LIN {X 69.907,Y 96.272,Z 65.686,A 180.000,B 0.000,C 180.000} C_DIS
LIN {X 69.876,Y 96.200,Z 65.684,A 180.000,B 0.000,C 180.000} C_DIS
LIN {X 69.842,Y 96.129,Z 65.681,A 180.000,B 0.000,C 180.000} C_DIS
LIN {X 69.807,Y 96.058,Z 65.678,A 180.000,B 0.000,C 180.000} C_DIS
LIN {X 69.735,Y 95.918,Z 65.673,A 180.000,B 0.000,C 180.000} C_DIS
LIN {X 69.664,Y 95.778,Z 65.668,A 180.000,B 0.000,C 180.000} C_DIS
LIN {X 69.628,Y 95.707,Z 65.665,A 180.000,B 0.000,C 180.000} C_DIS
LIN {X 69.592,Y 95.637,Z 65.662,A 180.000,B 0.000,C 180.000} C_DIS
LIN {X 69.557,Y 95.567,Z 65.660,A 180.000,B 0.000,C 180.000} C_DIS
LIN {X 69.521,Y 95.497,Z 65.657,A 180.000,B 0.000,C 180.000} C_DIS
LIN {X 69.483,Y 95.428,Z 65.655,A 180.000,B 0.000,C 180.000} C_DIS
LIN {X 69.443,Y 95.360,Z 65.652,A 180.000,B 0.000,C 180.000} C_DIS
LIN {X 69.403,Y 95.292,Z 65.650,A 180.000,B 0.000,C 180.000} C_DIS
LIN {X 69.323,Y 95.156,Z 65.645,A 180.000,B 0.000,C 180.000} C_DIS
LIN {X 69.243,Y 95.021,Z 65.640,A 180.000,B 0.000,C 180.000} C_DIS
LIN {X 69.163,Y 94.885,Z 65.635,A 180.000,B 0.000,C 180.000} C_DIS
LIN {X 69.081,Y 94.751,Z 65.630,A 180.000,B 0.000,C 180.000} C_DIS
LIN {X 68.992,Y 94.620,Z 65.625,A 180.000,B 0.000,C 180.000} C_DIS
LIN {X 68.904,Y 94.490,Z 65.621,A 180.000,B 0.000,C 180.000} C_DIS
LIN {X 68.815,Y 94.360,Z 65.616,A 180.000,B 0.000,C 180.000} C_DIS
LIN {X 68.727,Y 94.230,Z 65.612,A 180.000,B 0.000,C 180.000} C_DIS
LIN {X 68.636,Y 94.101,Z 65.607,A 180.000,B 0.000,C 180.000} C_DIS
LIN {X 68.540,Y 93.976,Z 65.603,A 180.000,B 0.000,C 180.000} C_DIS
LIN {X 68.444,Y 93.851,Z 65.598,A 180.000,B 0.000,C 180.000} C_DIS
LIN {X 68.347,Y 93.727,Z 65.594,A 180.000,B 0.000,C 180.000} C_DIS
LIN {X 68.251,Y 93.603,Z 65.590,A 180.000,B 0.000,C 180.000} C_DIS
LIN {X 68.152,Y 93.479,Z 65.586,A 180.000,B 0.000,C 180.000} C_DIS
LIN {X 68.049,Y 93.361,Z 65.582,A 180.000,B 0.000,C 180.000} C_DIS
LIN {X 67.945,Y 93.243,Z 65.578,A 180.000,B 0.000,C 180.000} C_DIS
LIN {X 67.840,Y 93.125,Z 65.574,A 180.000,B 0.000,C 180.000} C_DIS
LIN {X 67.736,Y 93.007,Z 65.571,A 180.000,B 0.000,C 180.000} C_DIS
LIN {X 67.630,Y 92.890,Z 65.567,A 180.000,B 0.000,C 180.000} C_DIS
LIN {X 67.519,Y 92.778,Z 65.563,A 180.000,B 0.000,C 180.000} C_DIS
LIN {X 67.408,Y 92.667,Z 65.560,A 180.000,B 0.000,C 180.000} C_DIS
LIN {X 67.297,Y 92.555,Z 65.556,A 180.000,B 0.000,C 180.000} C_DIS
LIN {X 67.185,Y 92.444,Z 65.553,A 180.000,B 0.000,C 180.000} C_DIS
LIN {X 67.072,Y 92.334,Z 65.550,A 180.000,B 0.000,C 180.000} C_DIS
LIN {X 66.955,Y 92.230,Z 65.547,A 180.000,B 0.000,C 180.000} C_DIS
LIN {X 66.837,Y 92.125,Z 65.544,A 180.000,B 0.000,C 180.000} C_DIS
LIN {X 66.718,Y 92.021,Z 65.541,A 180.000,B 0.000,C 180.000} C_DIS
LIN {X 66.600,Y 91.917,Z 65.538,A 180.000,B 0.000,C 180.000} C_DIS
LIN {X 66.481,Y 91.815,Z 65.535,A 180.000,B 0.000,C 180.000} C_DIS
LIN {X 66.357,Y 91.718,Z 65.532,A 180.000,B 0.000,C 180.000} C_DIS
LIN {X 66.232,Y 91.621,Z 65.530,A 180.000,B 0.000,C 180.000} C_DIS
LIN {X 66.108,Y 91.524,Z 65.527,A 180.000,B 0.000,C 180.000} C_DIS
LIN {X 65.858,Y 91.333,Z 65.523,A 180.000,B 0.000,C 180.000} C_DIS
LIN {X 65.597,Y 91.156,Z 65.518,A 180.000,B 0.000,C 180.000} C_DIS
LIN {X 65.337,Y 90.978,Z 65.515,A 180.000,B 0.000,C 180.000} C_DIS
LIN {X 65.070,Y 90.811,Z 65.511,A 180.000,B 0.000,C 180.000} C_DIS
LIN {X 64.799,Y 90.651,Z 65.508,A 180.000,B 0.000,C 180.000} C_DIS
LIN {X 64.527,Y 90.492,Z 65.506,A 180.000,B 0.000,C 180.000} C_DIS
LIN {X 64.247,Y 90.348,Z 65.504,A 180.000,B 0.000,C 180.000} C_DIS
LIN {X 63.966,Y 90.205,Z 65.502,A 180.000,B 0.000,C 180.000} C_DIS
LIN {X 63.680,Y 90.072,Z 65.501,A 180.000,B 0.000,C 180.000} C_DIS
LIN {X 63.391,Y 89.947,Z 65.500,A 180.000,B 0.000,C 180.000} C_DIS
LIN {X 63.141,Y 89.840,Z 65.500,A 180.000,B 0.000,C 180.000} C_DIS
; Cutting Move Starts
LIN {X 63.109,Y 89.827,Z 65.500,A 180.000,B 0.000,C 180.000} C_DIS
LIN {X 62.930,Y 89.762,Z 65.500,A 180.000,B 0.000,C 180.000} C_DIS
LIN {X 62.573,Y 89.633,Z 65.500,A 180.000,B 0.000,C 180.000} C_DIS
LIN {X 62.394,Y 89.569,Z 65.500,A 180.000,B 0.000,C 180.000} C_DIS
LIN {X 62.387,Y 89.567,Z 65.500,A 180.000,B 0.000,C 180.000} C_DIS
LIN {X 62.215,Y 89.516,Z 65.500,A 180.000,B 0.000,C 180.000} C_DIS
LIN {X 61.777,Y 89.388,Z 65.500,A 180.000,B 0.000,C 180.000} C_DIS
LIN {X 61.679,Y 89.360,Z 65.500,A 180.000,B 0.000,C 180.000} C_DIS
LIN {X 61.500,Y 89.316,Z 65.500,A 180.000,B 0.000,C 180.000} C_DIS
LIN {X 60.964,Y 89.196,Z 65.500,A 180.000,B 0.000,C 180.000} C_DIS
LIN {X 60.785,Y 89.161,Z 65.500,A 180.000,B 0.000,C 180.000} C_DIS
LIN {X 60.606,Y 89.132,Z 65.500,A 180.000,B 0.000,C 180.000} C_DIS
LIN {X 60.249,Y 89.076,Z 65.500,A 180.000,B 0.000,C 180.000} C_DIS
LIN {X 60.070,Y 89.049,Z 65.500,A 180.000,B 0.000,C 180.000} C_DIS
LIN {X 59.892,Y 89.031,Z 65.500,A 180.000,B 0.000,C 180.000} C_DIS
LIN {X 59.534,Y 88.997,Z 65.500,A 180.000,B 0.000,C 180.000} C_DIS
LIN {X 59.355,Y 88.980,Z 65.500,A 180.000,B 0.000,C 180.000} C_DIS
LIN {X 59.176,Y 88.970,Z 65.500,A 180.000,B 0.000,C 180.000} C_DIS
LIN {X 58.640,Y 88.953,Z 65.500,A 180.000,B 0.000,C 180.000} C_DIS
LIN {X 58.461,Y 88.950,Z 65.500,A 180.000,B 0.000,C 180.000} C_DIS
LIN {X 58.282,Y 88.956,Z 65.500,A 180.000,B 0.000,C 180.000} C_DIS
LIN {X 57.925,Y 88.967,Z 65.500,A 180.000,B 0.000,C 180.000} C_DIS
LIN {X 57.746,Y 88.973,Z 65.500,A 180.000,B 0.000,C 180.000} C_DIS
LIN {X 57.567,Y 88.987,Z 65.500,A 180.000,B 0.000,C 180.000} C_DIS
LIN {X 57.031,Y 89.038,Z 65.500,A 180.000,B 0.000,C 180.000} C_DIS
LIN {X 56.852,Y 89.060,Z 65.500,A 180.000,B 0.000,C 180.000} C_DIS
LIN {X 56.316,Y 89.145,Z 65.500,A 180.000,B 0.000,C 180.000} C_DIS
LIN {X 56.137,Y 89.174,Z 65.500,A 180.000,B 0.000,C 180.000} C_DIS
LIN {X 55.977,Y 89.209,Z 65.500,A 180.000,B 0.000,C 180.000} C_DIS
LIN {X 55.601,Y 89.293,Z 65.500,A 180.000,B 0.000,C 180.000} C_DIS
LIN {X 55.422,Y 89.334,Z 65.500,A 180.000,B 0.000,C 180.000} C_DIS
LIN {X 55.243,Y 89.382,Z 65.500,A 180.000,B 0.000,C 180.000} C_DIS
LIN {X 54.707,Y 89.538,Z 65.500,A 180.000,B 0.000,C 180.000} C_DIS
LIN {X 54.613,Y 89.567,Z 65.500,A 180.000,B 0.000,C 180.000} C_DIS
LIN {X 54.528,Y 89.597,Z 65.500,A 180.000,B 0.000,C 180.000} C_DIS
LIN {X 53.992,Y 89.790,Z 65.500,A 180.000,B 0.000,C 180.000} C_DIS
LIN {X 53.813,Y 89.859,Z 65.500,A 180.000,B 0.000,C 180.000} C_DIS
LIN {X 53.455,Y 90.014,Z 65.500,A 180.000,B 0.000,C 180.000} C_DIS
LIN {X 53.248,Y 90.103,Z 65.500,A 180.000,B 0.000,C 180.000} C_DIS
LIN {X 53.098,Y 90.173,Z 65.500,A 180.000,B 0.000,C 180.000} C_DIS
LIN {X 52.919,Y 90.264,Z 65.500,A 180.000,B 0.000,C 180.000} C_DIS
LIN {X 52.533,Y 90.461,Z 65.500,A 180.000,B 0.000,C 180.000} C_DIS
LIN {X 52.383,Y 90.543,Z 65.500,A 180.000,B 0.000,C 180.000} C_DIS
LIN {X 51.847,Y 90.860,Z 65.500,A 180.000,B 0.000,C 180.000} C_DIS
LIN {X 51.668,Y 90.975,Z 65.500,A 180.000,B 0.000,C 180.000} C_DIS
LIN {X 51.310,Y 91.218,Z 65.500,A 180.000,B 0.000,C 180.000} C_DIS
LIN {X 51.131,Y 91.341,Z 65.500,A 180.000,B 0.000,C 180.000} C_DIS
LIN {X 51.113,Y 91.355,Z 65.500,A 180.000,B 0.000,C 180.000} C_DIS
LIN {X 50.953,Y 91.478,Z 65.500,A 180.000,B 0.000,C 180.000} C_DIS
LIN {X 50.595,Y 91.755,Z 65.500,A 180.000,B 0.000,C 180.000} C_DIS
LIN {X 50.429,Y 91.891,Z 65.500,A 180.000,B 0.000,C 180.000} C_DIS
LIN {X 50.024,Y 92.249,Z 65.500,A 180.000,B 0.000,C 180.000} C_DIS
LIN {X 49.880,Y 92.379,Z 65.500,A 180.000,B 0.000,C 180.000} C_DIS
LIN {X 49.831,Y 92.427,Z 65.500,A 180.000,B 0.000,C 180.000} C_DIS
LIN {X 49.474,Y 92.785,Z 65.500,A 180.000,B 0.000,C 180.000} C_DIS
LIN {X 49.344,Y 92.917,Z 65.500,A 180.000,B 0.000,C 180.000} C_DIS
LIN {X 49.302,Y 92.964,Z 65.500,A 180.000,B 0.000,C 180.000} C_DIS
LIN {X 48.986,Y 93.321,Z 65.500,A 180.000,B 0.000,C 180.000} C_DIS
LIN {X 48.830,Y 93.500,Z 65.500,A 180.000,B 0.000,C 180.000} C_DIS
LIN {X 48.807,Y 93.528,Z 65.500,A 180.000,B 0.000,C 180.000} C_DIS
LIN {X 48.690,Y 93.679,Z 65.500,A 180.000,B 0.000,C 180.000} C_DIS
LIN {X 48.413,Y 94.036,Z 65.500,A 180.000,B 0.000,C 180.000} C_DIS
LIN {X 48.283,Y 94.215,Z 65.500,A 180.000,B 0.000,C 180.000} C_DIS
LIN {X 48.040,Y 94.573,Z 65.500,A 180.000,B 0.000,C 180.000} C_DIS
LIN {X 47.919,Y 94.751,Z 65.500,A 180.000,B 0.000,C 180.000} C_DIS
LIN {X 47.914,Y 94.760,Z 65.500,A 180.000,B 0.000,C 180.000} C_DIS
LIN {X 47.811,Y 94.930,Z 65.500,A 180.000,B 0.000,C 180.000} C_DIS
LIN {X 47.556,Y 95.361,Z 65.500,A 180.000,B 0.000,C 180.000} C_DIS
LIN {X 47.496,Y 95.466,Z 65.500,A 180.000,B 0.000,C 180.000} C_DIS
LIN {X 47.404,Y 95.645,Z 65.500,A 180.000,B 0.000,C 180.000} C_DIS
LIN {X 47.198,Y 96.048,Z 65.500,A 180.000,B 0.000,C 180.000} C_DIS
LIN {X 47.133,Y 96.181,Z 65.500,A 180.000,B 0.000,C 180.000} C_DIS
LIN {X 47.055,Y 96.360,Z 65.500,A 180.000,B 0.000,C 180.000} C_DIS
LIN {X 46.900,Y 96.718,Z 65.500,A 180.000,B 0.000,C 180.000} C_DIS
LIN {X 46.841,Y 96.856,Z 65.500,A 180.000,B 0.000,C 180.000} C_DIS
LIN {X 46.825,Y 96.897,Z 65.500,A 180.000,B 0.000,C 180.000} C_DIS
LIN {X 46.760,Y 97.075,Z 65.500,A 180.000,B 0.000,C 180.000} C_DIS
LIN {X 46.631,Y 97.433,Z 65.500,A 180.000,B 0.000,C 180.000} C_DIS
LIN {X 46.568,Y 97.612,Z 65.500,A 180.000,B 0.000,C 180.000} C_DIS
LIN {X 46.514,Y 97.790,Z 65.500,A 180.000,B 0.000,C 180.000} C_DIS
LIN {X 46.410,Y 98.148,Z 65.500,A 180.000,B 0.000,C 180.000} C_DIS
LIN {X 46.358,Y 98.327,Z 65.500,A 180.000,B 0.000,C 180.000} C_DIS
LIN {X 46.315,Y 98.505,Z 65.500,A 180.000,B 0.000,C 180.000} C_DIS
LIN {X 46.195,Y 99.042,Z 65.500,A 180.000,B 0.000,C 180.000} C_DIS
LIN {X 46.160,Y 99.221,Z 65.500,A 180.000,B 0.000,C 180.000} C_DIS
LIN {X 46.126,Y 99.434,Z 65.500,A 180.000,B 0.000,C 180.000} C_DIS
LIN {X 46.075,Y 99.757,Z 65.500,A 180.000,B 0.000,C 180.000} C_DIS
LIN {X 46.048,Y 99.936,Z 65.500,A 180.000,B 0.000,C 180.000} C_DIS
LIN {X 46.030,Y 100.114,Z 65.500,A 180.000,B 0.000,C 180.000} C_DIS
LIN {X 45.996,Y 100.472,Z 65.500,A 180.000,B 0.000,C 180.000} C_DIS
LIN {X 45.979,Y 100.651,Z 65.500,A 180.000,B 0.000,C 180.000} C_DIS
LIN {X 45.970,Y 100.829,Z 65.500,A 180.000,B 0.000,C 180.000} C_DIS
LIN {X 45.953,Y 101.366,Z 65.500,A 180.000,B 0.000,C 180.000} C_DIS
LIN {X 45.950,Y 101.545,Z 65.500,A 180.000,B 0.000,C 180.000} C_DIS
LIN {X 45.956,Y 101.723,Z 65.500,A 180.000,B 0.000,C 180.000} C_DIS
LIN {X 45.967,Y 102.081,Z 65.500,A 180.000,B 0.000,C 180.000} C_DIS
LIN {X 45.973,Y 102.260,Z 65.500,A 180.000,B 0.000,C 180.000} C_DIS
LIN {X 45.988,Y 102.438,Z 65.500,A 180.000,B 0.000,C 180.000} C_DIS
LIN {X 46.038,Y 102.975,Z 65.500,A 180.000,B 0.000,C 180.000} C_DIS
LIN {X 46.060,Y 103.153,Z 65.500,A 180.000,B 0.000,C 180.000} C_DIS
LIN {X 46.145,Y 103.690,Z 65.500,A 180.000,B 0.000,C 180.000} C_DIS
LIN {X 46.176,Y 103.869,Z 65.500,A 180.000,B 0.000,C 180.000} C_DIS
LIN {X 46.215,Y 104.047,Z 65.500,A 180.000,B 0.000,C 180.000} C_DIS
LIN {X 46.305,Y 104.449,Z 65.500,A 180.000,B 0.000,C 180.000} C_DIS
LIN {X 46.335,Y 104.584,Z 65.500,A 180.000,B 0.000,C 180.000} C_DIS
LIN {X 46.384,Y 104.762,Z 65.500,A 180.000,B 0.000,C 180.000} C_DIS
LIN {X 46.540,Y 105.299,Z 65.500,A 180.000,B 0.000,C 180.000} C_DIS
LIN {X 46.599,Y 105.477,Z 65.500,A 180.000,B 0.000,C 180.000} C_DIS
LIN {X 46.792,Y 106.014,Z 65.500,A 180.000,B 0.000,C 180.000} C_DIS
LIN {X 46.841,Y 106.144,Z 65.500,A 180.000,B 0.000,C 180.000} C_DIS
LIN {X 46.861,Y 106.193,Z 65.500,A 180.000,B 0.000,C 180.000} C_DIS
LIN {X 47.093,Y 106.729,Z 65.500,A 180.000,B 0.000,C 180.000} C_DIS
LIN {X 47.176,Y 106.908,Z 65.500,A 180.000,B 0.000,C 180.000} C_DIS
LIN {X 47.198,Y 106.952,Z 65.500,A 180.000,B 0.000,C 180.000} C_DIS
LIN {X 47.449,Y 107.444,Z 65.500,A 180.000,B 0.000,C 180.000} C_DIS
LIN {X 47.546,Y 107.623,Z 65.500,A 180.000,B 0.000,C 180.000} C_DIS
LIN {X 47.863,Y 108.159,Z 65.500,A 180.000,B 0.000,C 180.000} C_DIS
LIN {X 47.914,Y 108.240,Z 65.500,A 180.000,B 0.000,C 180.000} C_DIS
LIN {X 47.979,Y 108.338,Z 65.500,A 180.000,B 0.000,C 180.000} C_DIS
LIN {X 48.271,Y 108.767,Z 65.500,A 180.000,B 0.000,C 180.000} C_DIS
LIN {X 48.345,Y 108.874,Z 65.500,A 180.000,B 0.000,C 180.000} C_DIS
LIN {X 48.450,Y 109.012,Z 65.500,A 180.000,B 0.000,C 180.000} C_DIS
LIN {X 48.759,Y 109.410,Z 65.500,A 180.000,B 0.000,C 180.000} C_DIS
LIN {X 48.807,Y 109.472,Z 65.500,A 180.000,B 0.000,C 180.000} C_DIS
LIN {X 48.907,Y 109.589,Z 65.500,A 180.000,B 0.000,C 180.000} C_DIS
LIN {X 49.223,Y 109.947,Z 65.500,A 180.000,B 0.000,C 180.000} C_DIS
LIN {X 49.344,Y 110.083,Z 65.500,A 180.000,B 0.000,C 180.000} C_DIS
LIN {X 49.384,Y 110.126,Z 65.500,A 180.000,B 0.000,C 180.000} C_DIS
LIN {X 49.523,Y 110.264,Z 65.500,A 180.000,B 0.000,C 180.000} C_DIS
LIN {X 49.742,Y 110.483,Z 65.500,A 180.000,B 0.000,C 180.000} C_DIS
LIN {X 49.880,Y 110.621,Z 65.500,A 180.000,B 0.000,C 180.000} C_DIS
LIN {X 49.923,Y 110.662,Z 65.500,A 180.000,B 0.000,C 180.000} C_DIS
LIN {X 50.059,Y 110.782,Z 65.500,A 180.000,B 0.000,C 180.000} C_DIS
LIN {X 50.416,Y 111.098,Z 65.500,A 180.000,B 0.000,C 180.000} C_DIS
LIN {X 50.535,Y 111.198,Z 65.500,A 180.000,B 0.000,C 180.000} C_DIS
LIN {X 50.595,Y 111.245,Z 65.500,A 180.000,B 0.000,C 180.000} C_DIS
LIN {X 50.996,Y 111.556,Z 65.500,A 180.000,B 0.000,C 180.000} C_DIS
LIN {X 51.131,Y 111.659,Z 65.500,A 180.000,B 0.000,C 180.000} C_DIS
LIN {X 51.241,Y 111.734,Z 65.500,A 180.000,B 0.000,C 180.000} C_DIS
LIN {X 51.668,Y 112.025,Z 65.500,A 180.000,B 0.000,C 180.000} C_DIS
LIN {X 51.769,Y 112.092,Z 65.500,A 180.000,B 0.000,C 180.000} C_DIS
LIN {X 51.847,Y 112.140,Z 65.500,A 180.000,B 0.000,C 180.000} C_DIS
LIN {X 52.383,Y 112.457,Z 65.500,A 180.000,B 0.000,C 180.000} C_DIS
LIN {X 52.562,Y 112.554,Z 65.500,A 180.000,B 0.000,C 180.000} C_DIS
LIN {X 53.059,Y 112.807,Z 65.500,A 180.000,B 0.000,C 180.000} C_DIS
LIN {X 53.098,Y 112.827,Z 65.500,A 180.000,B 0.000,C 180.000} C_DIS
LIN {X 53.277,Y 112.909,Z 65.500,A 180.000,B 0.000,C 180.000} C_DIS
LIN {X 53.813,Y 113.141,Z 65.500,A 180.000,B 0.000,C 180.000} C_DIS
LIN {X 53.870,Y 113.165,Z 65.500,A 180.000,B 0.000,C 180.000} C_DIS
LIN {X 53.992,Y 113.210,Z 65.500,A 180.000,B 0.000,C 180.000} C_DIS
LIN {X 54.528,Y 113.403,Z 65.500,A 180.000,B 0.000,C 180.000} C_DIS
LIN {X 54.707,Y 113.462,Z 65.500,A 180.000,B 0.000,C 180.000} C_DIS
LIN {X 55.243,Y 113.618,Z 65.500,A 180.000,B 0.000,C 180.000} C_DIS
LIN {X 55.422,Y 113.666,Z 65.500,A 180.000,B 0.000,C 180.000} C_DIS
LIN {X 55.575,Y 113.701,Z 65.500,A 180.000,B 0.000,C 180.000} C_DIS
LIN {X 55.958,Y 113.786,Z 65.500,A 180.000,B 0.000,C 180.000} C_DIS
LIN {X 56.056,Y 113.808,Z 65.500,A 180.000,B 0.000,C 180.000} C_DIS
LIN {X 56.137,Y 113.826,Z 65.500,A 180.000,B 0.000,C 180.000} C_DIS
LIN {X 56.316,Y 113.855,Z 65.500,A 180.000,B 0.000,C 180.000} C_DIS
LIN {X 56.852,Y 113.940,Z 65.500,A 180.000,B 0.000,C 180.000} C_DIS
LIN {X 57.031,Y 113.962,Z 65.500,A 180.000,B 0.000,C 180.000} C_DIS
LIN {X 57.567,Y 114.013,Z 65.500,A 180.000,B 0.000,C 180.000} C_DIS
LIN {X 57.746,Y 114.027,Z 65.500,A 180.000,B 0.000,C 180.000} C_DIS
LIN {X 57.925,Y 114.033,Z 65.500,A 180.000,B 0.000,C 180.000} C_DIS
LIN {X 58.282,Y 114.044,Z 65.500,A 180.000,B 0.000,C 180.000} C_DIS
LIN {X 58.461,Y 114.050,Z 65.500,A 180.000,B 0.000,C 180.000} C_DIS
LIN {X 58.640,Y 114.047,Z 65.500,A 180.000,B 0.000,C 180.000} C_DIS
LIN {X 59.176,Y 114.030,Z 65.500,A 180.000,B 0.000,C 180.000} C_DIS
LIN {X 59.355,Y 114.020,Z 65.500,A 180.000,B 0.000,C 180.000} C_DIS
LIN {X 59.534,Y 114.003,Z 65.500,A 180.000,B 0.000,C 180.000} C_DIS
LIN {X 59.891,Y 113.969,Z 65.500,A 180.000,B 0.000,C 180.000} C_DIS
LIN {X 60.070,Y 113.951,Z 65.500,A 180.000,B 0.000,C 180.000} C_DIS
LIN {X 60.249,Y 113.924,Z 65.500,A 180.000,B 0.000,C 180.000} C_DIS
LIN {X 60.606,Y 113.868,Z 65.500,A 180.000,B 0.000,C 180.000} C_DIS
LIN {X 60.785,Y 113.839,Z 65.500,A 180.000,B 0.000,C 180.000} C_DIS
LIN {X 60.964,Y 113.804,Z 65.500,A 180.000,B 0.000,C 180.000} C_DIS
LIN {X 61.500,Y 113.684,Z 65.500,A 180.000,B 0.000,C 180.000} C_DIS
LIN {X 61.679,Y 113.640,Z 65.500,A 180.000,B 0.000,C 180.000} C_DIS
LIN {X 61.858,Y 113.588,Z 65.500,A 180.000,B 0.000,C 180.000} C_DIS
LIN {X 62.215,Y 113.484,Z 65.500,A 180.000,B 0.000,C 180.000} C_DIS
LIN {X 62.394,Y 113.431,Z 65.500,A 180.000,B 0.000,C 180.000} C_DIS
LIN {X 62.573,Y 113.367,Z 65.500,A 180.000,B 0.000,C 180.000} C_DIS
LIN {X 62.930,Y 113.238,Z 65.500,A 180.000,B 0.000,C 180.000} C_DIS
LIN {X 63.109,Y 113.173,Z 65.500,A 180.000,B 0.000,C 180.000} C_DIS
LIN {X 63.130,Y 113.165,Z 65.500,A 180.000,B 0.000,C 180.000} C_DIS
LIN {X 63.288,Y 113.097,Z 65.500,A 180.000,B 0.000,C 180.000} C_DIS
LIN {X 63.645,Y 112.943,Z 65.500,A 180.000,B 0.000,C 180.000} C_DIS
LIN {X 63.824,Y 112.865,Z 65.500,A 180.000,B 0.000,C 180.000} C_DIS
LIN {X 63.941,Y 112.807,Z 65.500,A 180.000,B 0.000,C 180.000} C_DIS
LIN {X 64.360,Y 112.594,Z 65.500,A 180.000,B 0.000,C 180.000} C_DIS
LIN {X 64.539,Y 112.501,Z 65.500,A 180.000,B 0.000,C 180.000} C_DIS
LIN {X 64.630,Y 112.450,Z 65.500,A 180.000,B 0.000,C 180.000} C_DIS
LIN {X 65.075,Y 112.186,Z 65.500,A 180.000,B 0.000,C 180.000} C_DIS
LIN {X 65.231,Y 112.092,Z 65.500,A 180.000,B 0.000,C 180.000} C_DIS
LIN {X 65.254,Y 112.077,Z 65.500,A 180.000,B 0.000,C 180.000} C_DIS
LIN {X 65.433,Y 111.956,Z 65.500,A 180.000,B 0.000,C 180.000} C_DIS
LIN {X 65.791,Y 111.713,Z 65.500,A 180.000,B 0.000,C 180.000} C_DIS
LIN {X 65.969,Y 111.583,Z 65.500,A 180.000,B 0.000,C 180.000} C_DIS
LIN {X 66.327,Y 111.306,Z 65.500,A 180.000,B 0.000,C 180.000} C_DIS
LIN {X 66.465,Y 111.198,Z 65.500,A 180.000,B 0.000,C 180.000} C_DIS
LIN {X 66.506,Y 111.165,Z 65.500,A 180.000,B 0.000,C 180.000} C_DIS
LIN {X 66.672,Y 111.019,Z 65.500,A 180.000,B 0.000,C 180.000} C_DIS
LIN {X 66.875,Y 110.841,Z 65.500,A 180.000,B 0.000,C 180.000} C_DIS
LIN {X 67.042,Y 110.693,Z 65.500,A 180.000,B 0.000,C 180.000} C_DIS
LIN {X 67.077,Y 110.662,Z 65.500,A 180.000,B 0.000,C 180.000} C_DIS
LIN {X 67.221,Y 110.521,Z 65.500,A 180.000,B 0.000,C 180.000} C_DIS
LIN {X 67.578,Y 110.163,Z 65.500,A 180.000,B 0.000,C 180.000} C_DIS
LIN {X 67.616,Y 110.126,Z 65.500,A 180.000,B 0.000,C 180.000} C_DIS
LIN {X 67.757,Y 109.970,Z 65.500,A 180.000,B 0.000,C 180.000} C_DIS
LIN {X 68.115,Y 109.564,Z 65.500,A 180.000,B 0.000,C 180.000} C_DIS
LIN {X 68.241,Y 109.410,Z 65.500,A 180.000,B 0.000,C 180.000} C_DIS
LIN {X 68.518,Y 109.053,Z 65.500,A 180.000,B 0.000,C 180.000} C_DIS
LIN {X 68.651,Y 108.880,Z 65.500,A 180.000,B 0.000,C 180.000} C_DIS
LIN {X 68.655,Y 108.874,Z 65.500,A 180.000,B 0.000,C 180.000} C_DIS
LIN {X 68.778,Y 108.695,Z 65.500,A 180.000,B 0.000,C 180.000} C_DIS
LIN {X 69.021,Y 108.338,Z 65.500,A 180.000,B 0.000,C 180.000} C_DIS
LIN {X 69.137,Y 108.159,Z 65.500,A 180.000,B 0.000,C 180.000} C_DIS
LIN {X 69.454,Y 107.623,Z 65.500,A 180.000,B 0.000,C 180.000} C_DIS
LIN {X 69.545,Y 107.456,Z 65.500,A 180.000,B 0.000,C 180.000} C_DIS
LIN {X 69.733,Y 107.086,Z 65.500,A 180.000,B 0.000,C 180.000} C_DIS
LIN {X 69.824,Y 106.908,Z 65.500,A 180.000,B 0.000,C 180.000} C_DIS
LIN {X 69.902,Y 106.739,Z 65.500,A 180.000,B 0.000,C 180.000} C_DIS
LIN {X 70.139,Y 106.193,Z 65.500,A 180.000,B 0.000,C 180.000} C_DIS
LIN {X 70.208,Y 106.014,Z 65.500,A 180.000,B 0.000,C 180.000} C_DIS
LIN {X 70.401,Y 105.477,Z 65.500,A 180.000,B 0.000,C 180.000} C_DIS
LIN {X 70.439,Y 105.369,Z 65.500,A 180.000,B 0.000,C 180.000} C_DIS
LIN {X 70.460,Y 105.299,Z 65.500,A 180.000,B 0.000,C 180.000} C_DIS
LIN {X 70.617,Y 104.758,Z 65.500,A 180.000,B 0.000,C 180.000} C_DIS
LIN {X 70.665,Y 104.584,Z 65.500,A 180.000,B 0.000,C 180.000} C_DIS
LIN {X 70.705,Y 104.405,Z 65.500,A 180.000,B 0.000,C 180.000} C_DIS
LIN {X 70.796,Y 103.999,Z 65.500,A 180.000,B 0.000,C 180.000} C_DIS
LIN {X 70.824,Y 103.869,Z 65.500,A 180.000,B 0.000,C 180.000} C_DIS
LIN {X 70.855,Y 103.690,Z 65.500,A 180.000,B 0.000,C 180.000} C_DIS
LIN {X 70.940,Y 103.153,Z 65.500,A 180.000,B 0.000,C 180.000} C_DIS
LIN {X 70.962,Y 102.975,Z 65.500,A 180.000,B 0.000,C 180.000} C_DIS
LIN {X 71.012,Y 102.438,Z 65.500,A 180.000,B 0.000,C 180.000} C_DIS
LIN {X 71.027,Y 102.260,Z 65.500,A 180.000,B 0.000,C 180.000} C_DIS
LIN {X 71.033,Y 102.081,Z 65.500,A 180.000,B 0.000,C 180.000} C_DIS
LIN {X 71.044,Y 101.723,Z 65.500,A 180.000,B 0.000,C 180.000} C_DIS
LIN {X 71.050,Y 101.545,Z 65.500,A 180.000,B 0.000,C 180.000} C_DIS
LIN {X 71.047,Y 101.366,Z 65.500,A 180.000,B 0.000,C 180.000} C_DIS
LIN {X 71.030,Y 100.829,Z 65.500,A 180.000,B 0.000,C 180.000} C_DIS
LIN {X 71.021,Y 100.651,Z 65.500,A 180.000,B 0.000,C 180.000} C_DIS
LIN {X 71.004,Y 100.472,Z 65.500,A 180.000,B 0.000,C 180.000} C_DIS
LIN {X 70.970,Y 100.114,Z 65.500,A 180.000,B 0.000,C 180.000} C_DIS
LIN {X 70.952,Y 99.936,Z 65.500,A 180.000,B 0.000,C 180.000} C_DIS
LIN {X 70.925,Y 99.757,Z 65.500,A 180.000,B 0.000,C 180.000} C_DIS
LIN {X 70.840,Y 99.221,Z 65.500,A 180.000,B 0.000,C 180.000} C_DIS
LIN {X 70.805,Y 99.042,Z 65.500,A 180.000,B 0.000,C 180.000} C_DIS
LIN {X 70.718,Y 98.654,Z 65.500,A 180.000,B 0.000,C 180.000} C_DIS
LIN {X 70.685,Y 98.505,Z 65.500,A 180.000,B 0.000,C 180.000} C_DIS
LIN {X 70.642,Y 98.327,Z 65.500,A 180.000,B 0.000,C 180.000} C_DIS
LIN {X 70.617,Y 98.242,Z 65.500,A 180.000,B 0.000,C 180.000} C_DIS
LIN {X 70.486,Y 97.790,Z 65.500,A 180.000,B 0.000,C 180.000} C_DIS
LIN {X 70.439,Y 97.631,Z 65.500,A 180.000,B 0.000,C 180.000} C_DIS
LIN {X 70.432,Y 97.612,Z 65.500,A 180.000,B 0.000,C 180.000} C_DIS
LIN {X 70.369,Y 97.433,Z 65.500,A 180.000,B 0.000,C 180.000} C_DIS
LIN {X 70.240,Y 97.075,Z 65.500,A 180.000,B 0.000,C 180.000} C_DIS
LIN {X 70.175,Y 96.897,Z 65.500,A 180.000,B 0.000,C 180.000} C_DIS
LIN {X 70.100,Y 96.718,Z 65.500,A 180.000,B 0.000,C 180.000} C_DIS
LIN {X 69.902,Y 96.261,Z 65.500,A 180.000,B 0.000,C 180.000} C_DIS
LIN {X 69.867,Y 96.181,Z 65.500,A 180.000,B 0.000,C 180.000} C_DIS
LIN {X 69.779,Y 96.003,Z 65.500,A 180.000,B 0.000,C 180.000} C_DIS
LIN {X 69.545,Y 95.544,Z 65.500,A 180.000,B 0.000,C 180.000} C_DIS
LIN {X 69.504,Y 95.466,Z 65.500,A 180.000,B 0.000,C 180.000} C_DIS
LIN {X 69.401,Y 95.288,Z 65.500,A 180.000,B 0.000,C 180.000} C_DIS
LIN {X 69.187,Y 94.927,Z 65.500,A 180.000,B 0.000,C 180.000} C_DIS
LIN {X 69.081,Y 94.751,Z 65.500,A 180.000,B 0.000,C 180.000} C_DIS
LIN {X 69.008,Y 94.644,Z 65.500,A 180.000,B 0.000,C 180.000} C_DIS
LIN {X 68.717,Y 94.215,Z 65.500,A 180.000,B 0.000,C 180.000} C_DIS
LIN {X 68.651,Y 94.120,Z 65.500,A 180.000,B 0.000,C 180.000} C_DIS
LIN {X 68.587,Y 94.036,Z 65.500,A 180.000,B 0.000,C 180.000} C_DIS
LIN {X 68.293,Y 93.657,Z 65.500,A 180.000,B 0.000,C 180.000} C_DIS
LIN {X 68.170,Y 93.500,Z 65.500,A 180.000,B 0.000,C 180.000} C_DIS
LIN {X 68.115,Y 93.436,Z 65.500,A 180.000,B 0.000,C 180.000} C_DIS
LIN {X 67.698,Y 92.964,Z 65.500,A 180.000,B 0.000,C 180.000} C_DIS
LIN {X 67.578,Y 92.837,Z 65.500,A 180.000,B 0.000,C 180.000} C_DIS
LIN {X 67.169,Y 92.427,Z 65.500,A 180.000,B 0.000,C 180.000} C_DIS
LIN {X 67.042,Y 92.307,Z 65.500,A 180.000,B 0.000,C 180.000} C_DIS
LIN {X 66.976,Y 92.249,Z 65.500,A 180.000,B 0.000,C 180.000} C_DIS
LIN {X 66.571,Y 91.891,Z 65.500,A 180.000,B 0.000,C 180.000} C_DIS
LIN {X 66.506,Y 91.835,Z 65.500,A 180.000,B 0.000,C 180.000} C_DIS
LIN {X 66.350,Y 91.712,Z 65.500,A 180.000,B 0.000,C 180.000} C_DIS
LIN {X 65.969,Y 91.417,Z 65.500,A 180.000,B 0.000,C 180.000} C_DIS
LIN {X 65.887,Y 91.355,Z 65.500,A 180.000,B 0.000,C 180.000} C_DIS
LIN {X 65.791,Y 91.287,Z 65.500,A 180.000,B 0.000,C 180.000} C_DIS
LIN {X 65.364,Y 90.997,Z 65.500,A 180.000,B 0.000,C 180.000} C_DIS
LIN {X 65.254,Y 90.923,Z 65.500,A 180.000,B 0.000,C 180.000} C_DIS
LIN {X 65.083,Y 90.818,Z 65.500,A 180.000,B 0.000,C 180.000} C_DIS
LIN {X 64.718,Y 90.603,Z 65.500,A 180.000,B 0.000,C 180.000} C_DIS
LIN {X 64.539,Y 90.499,Z 65.500,A 180.000,B 0.000,C 180.000} C_DIS
LIN {X 64.467,Y 90.461,Z 65.500,A 180.000,B 0.000,C 180.000} C_DIS
LIN {X 64.003,Y 90.224,Z 65.500,A 180.000,B 0.000,C 180.000} C_DIS
LIN {X 63.824,Y 90.135,Z 65.500,A 180.000,B 0.000,C 180.000} C_DIS
LIN {X 63.752,Y 90.103,Z 65.500,A 180.000,B 0.000,C 180.000} C_DIS
LIN {X 63.288,Y 89.903,Z 65.500,A 180.000,B 0.000,C 180.000} C_DIS
LIN {X 63.141,Y 89.840,Z 65.500,A 180.000,B 0.000,C 180.000} C_DIS
; Link Move Starts
LIN {X 62.845,Y 89.731,Z 65.500,A 180.000,B 0.000,C 180.000} C_DIS
LIN {X 62.549,Y 89.624,Z 65.499,A 180.000,B 0.000,C 180.000} C_DIS
LIN {X 62.250,Y 89.526,Z 65.498,A 180.000,B 0.000,C 180.000} C_DIS
LIN {X 61.947,Y 89.438,Z 65.496,A 180.000,B 0.000,C 180.000} C_DIS
LIN {X 61.645,Y 89.350,Z 65.494,A 180.000,B 0.000,C 180.000} C_DIS
LIN {X 61.338,Y 89.280,Z 65.491,A 180.000,B 0.000,C 180.000} C_DIS
LIN {X 61.030,Y 89.211,Z 65.488,A 180.000,B 0.000,C 180.000} C_DIS
LIN {X 60.721,Y 89.150,Z 65.485,A 180.000,B 0.000,C 180.000} C_DIS
LIN {X 60.410,Y 89.101,Z 65.481,A 180.000,B 0.000,C 180.000} C_DIS
LIN {X 60.099,Y 89.052,Z 65.477,A 180.000,B 0.000,C 180.000} C_DIS
LIN {X 59.786,Y 89.021,Z 65.472,A 180.000,B 0.000,C 180.000} C_DIS
LIN {X 59.629,Y 89.006,Z 65.469,A 180.000,B 0.000,C 180.000} C_DIS
LIN {X 59.472,Y 88.991,Z 65.467,A 180.000,B 0.000,C 180.000} C_DIS
LIN {X 59.315,Y 88.977,Z 65.464,A 180.000,B 0.000,C 180.000} C_DIS
LIN {X 59.158,Y 88.969,Z 65.461,A 180.000,B 0.000,C 180.000} C_DIS
LIN {X 59.000,Y 88.964,Z 65.459,A 180.000,B 0.000,C 180.000} C_DIS
LIN {X 58.843,Y 88.960,Z 65.456,A 180.000,B 0.000,C 180.000} C_DIS
LIN {X 58.685,Y 88.955,Z 65.452,A 180.000,B 0.000,C 180.000} C_DIS
LIN {X 58.528,Y 88.950,Z 65.449,A 180.000,B 0.000,C 180.000} C_DIS
LIN {X 58.371,Y 88.953,Z 65.446,A 180.000,B 0.000,C 180.000} C_DIS
LIN {X 58.213,Y 88.958,Z 65.443,A 180.000,B 0.000,C 180.000} C_DIS
LIN {X 58.056,Y 88.963,Z 65.439,A 180.000,B 0.000,C 180.000} C_DIS
LIN {X 57.898,Y 88.968,Z 65.436,A 180.000,B 0.000,C 180.000} C_DIS
LIN {X 57.741,Y 88.973,Z 65.432,A 180.000,B 0.000,C 180.000} C_DIS
LIN {X 57.584,Y 88.986,Z 65.428,A 180.000,B 0.000,C 180.000} C_DIS
LIN {X 57.427,Y 89.000,Z 65.425,A 180.000,B 0.000,C 180.000} C_DIS
LIN {X 57.270,Y 89.015,Z 65.421,A 180.000,B 0.000,C 180.000} C_DIS
LIN {X 57.113,Y 89.030,Z 65.417,A 180.000,B 0.000,C 180.000} C_DIS
LIN {X 56.957,Y 89.045,Z 65.413,A 180.000,B 0.000,C 180.000} C_DIS
LIN {X 56.801,Y 89.068,Z 65.409,A 180.000,B 0.000,C 180.000} C_DIS
LIN {X 56.645,Y 89.092,Z 65.405,A 180.000,B 0.000,C 180.000} C_DIS
LIN {X 56.490,Y 89.117,Z 65.400,A 180.000,B 0.000,C 180.000} C_DIS
LIN {X 56.334,Y 89.142,Z 65.396,A 180.000,B 0.000,C 180.000} C_DIS
LIN {X 56.179,Y 89.167,Z 65.392,A 180.000,B 0.000,C 180.000} C_DIS
LIN {X 56.024,Y 89.199,Z 65.387,A 180.000,B 0.000,C 180.000} C_DIS
LIN {X 55.871,Y 89.233,Z 65.383,A 180.000,B 0.000,C 180.000} C_DIS
LIN {X 55.717,Y 89.267,Z 65.378,A 180.000,B 0.000,C 180.000} C_DIS
LIN {X 55.563,Y 89.302,Z 65.373,A 180.000,B 0.000,C 180.000} C_DIS
LIN {X 55.410,Y 89.337,Z 65.369,A 180.000,B 0.000,C 180.000} C_DIS
LIN {X 55.258,Y 89.378,Z 65.364,A 180.000,B 0.000,C 180.000} C_DIS
LIN {X 55.107,Y 89.422,Z 65.359,A 180.000,B 0.000,C 180.000} C_DIS
LIN {X 54.955,Y 89.466,Z 65.354,A 180.000,B 0.000,C 180.000} C_DIS
LIN {X 54.880,Y 89.488,Z 65.351,A 180.000,B 0.000,C 180.000} C_DIS
LIN {X 54.804,Y 89.510,Z 65.349,A 180.000,B 0.000,C 180.000} C_DIS
LIN {X 54.728,Y 89.532,Z 65.346,A 180.000,B 0.000,C 180.000} C_DIS
LIN {X 54.653,Y 89.554,Z 65.344,A 180.000,B 0.000,C 180.000} C_DIS
LIN {X 54.578,Y 89.579,Z 65.341,A 180.000,B 0.000,C 180.000} C_DIS
LIN {X 54.504,Y 89.605,Z 65.339,A 180.000,B 0.000,C 180.000} C_DIS
LIN {X 54.430,Y 89.632,Z 65.336,A 180.000,B 0.000,C 180.000} C_DIS
LIN {X 54.282,Y 89.685,Z 65.331,A 180.000,B 0.000,C 180.000} C_DIS
LIN {X 54.133,Y 89.739,Z 65.325,A 180.000,B 0.000,C 180.000} C_DIS
LIN {X 53.985,Y 89.792,Z 65.320,A 180.000,B 0.000,C 180.000} C_DIS
LIN {X 53.911,Y 89.819,Z 65.317,A 180.000,B 0.000,C 180.000} C_DIS
LIN {X 53.838,Y 89.848,Z 65.315,A 180.000,B 0.000,C 180.000} C_DIS
LIN {X 53.766,Y 89.879,Z 65.312,A 180.000,B 0.000,C 180.000} C_DIS
LIN {X 53.477,Y 90.005,Z 65.301,A 180.000,B 0.000,C 180.000} C_DIS
LIN {X 53.260,Y 90.098,Z 65.293,A 180.000,B 0.000,C 180.000} C_DIS
LIN {X 53.188,Y 90.130,Z 65.290,A 180.000,B 0.000,C 180.000} C_DIS
LIN {X 53.117,Y 90.164,Z 65.287,A 180.000,B 0.000,C 180.000} C_DIS
LIN {X 53.046,Y 90.199,Z 65.285,A 180.000,B 0.000,C 180.000} C_DIS
LIN {X 52.906,Y 90.271,Z 65.279,A 180.000,B 0.000,C 180.000} C_DIS
LIN {X 52.695,Y 90.378,Z 65.271,A 180.000,B 0.000,C 180.000} C_DIS
LIN {X 52.555,Y 90.449,Z 65.265,A 180.000,B 0.000,C 180.000} C_DIS
LIN {X 52.485,Y 90.486,Z 65.263,A 180.000,B 0.000,C 180.000} C_DIS
LIN {X 52.416,Y 90.524,Z 65.260,A 180.000,B 0.000,C 180.000} C_DIS
LIN {X 52.348,Y 90.563,Z 65.257,A 180.000,B 0.000,C 180.000} C_DIS
LIN {X 52.145,Y 90.684,Z 65.249,A 180.000,B 0.000,C 180.000} C_DIS
LIN {X 52.009,Y 90.764,Z 65.243,A 180.000,B 0.000,C 180.000} C_DIS
LIN {X 51.942,Y 90.804,Z 65.241,A 180.000,B 0.000,C 180.000} C_DIS
LIN {X 51.874,Y 90.844,Z 65.238,A 180.000,B 0.000,C 180.000} C_DIS
LIN {X 51.806,Y 90.884,Z 65.235,A 180.000,B 0.000,C 180.000} C_DIS
LIN {X 51.740,Y 90.927,Z 65.232,A 180.000,B 0.000,C 180.000} C_DIS
LIN {X 51.674,Y 90.971,Z 65.230,A 180.000,B 0.000,C 180.000} C_DIS
LIN {X 51.544,Y 91.059,Z 65.224,A 180.000,B 0.000,C 180.000} C_DIS
LIN {X 51.218,Y 91.281,Z 65.210,A 180.000,B 0.000,C 180.000} C_DIS
LIN {X 51.154,Y 91.325,Z 65.208,A 180.000,B 0.000,C 180.000} C_DIS
LIN {X 51.090,Y 91.372,Z 65.205,A 180.000,B 0.000,C 180.000} C_DIS
LIN {X 51.027,Y 91.420,Z 65.202,A 180.000,B 0.000,C 180.000} C_DIS
LIN {X 50.654,Y 91.709,Z 65.186,A 180.000,B 0.000,C 180.000} C_DIS
LIN {X 50.592,Y 91.757,Z 65.183,A 180.000,B 0.000,C 180.000} C_DIS
LIN {X 50.530,Y 91.806,Z 65.180,A 180.000,B 0.000,C 180.000} C_DIS
LIN {X 50.469,Y 91.856,Z 65.177,A 180.000,B 0.000,C 180.000} C_DIS
LIN {X 50.410,Y 91.908,Z 65.175,A 180.000,B 0.000,C 180.000} C_DIS
LIN {X 50.292,Y 92.012,Z 65.169,A 180.000,B 0.000,C 180.000} C_DIS
LIN {X 49.996,Y 92.273,Z 65.155,A 180.000,B 0.000,C 180.000} C_DIS
LIN {X 49.938,Y 92.325,Z 65.153,A 180.000,B 0.000,C 180.000} C_DIS
LIN {X 49.880,Y 92.379,Z 65.150,A 180.000,B 0.000,C 180.000} C_DIS
LIN {X 49.824,Y 92.434,Z 65.147,A 180.000,B 0.000,C 180.000} C_DIS
LIN {X 49.434,Y 92.824,Z 65.128,A 180.000,B 0.000,C 180.000} C_DIS
LIN {X 49.379,Y 92.880,Z 65.125,A 180.000,B 0.000,C 180.000} C_DIS
LIN {X 49.325,Y 92.937,Z 65.122,A 180.000,B 0.000,C 180.000} C_DIS
LIN {X 49.273,Y 92.996,Z 65.120,A 180.000,B 0.000,C 180.000} C_DIS
LIN {X 49.117,Y 93.174,Z 65.111,A 180.000,B 0.000,C 180.000} C_DIS
LIN {X 49.012,Y 93.292,Z 65.106,A 180.000,B 0.000,C 180.000} C_DIS
LIN {X 48.908,Y 93.410,Z 65.100,A 180.000,B 0.000,C 180.000} C_DIS
LIN {X 48.856,Y 93.469,Z 65.098,A 180.000,B 0.000,C 180.000} C_DIS
LIN {X 48.806,Y 93.530,Z 65.095,A 180.000,B 0.000,C 180.000} C_DIS
LIN {X 48.758,Y 93.592,Z 65.092,A 180.000,B 0.000,C 180.000} C_DIS
LIN {X 48.420,Y 94.027,Z 65.073,A 180.000,B 0.000,C 180.000} C_DIS
LIN {X 48.372,Y 94.090,Z 65.070,A 180.000,B 0.000,C 180.000} C_DIS
LIN {X 48.325,Y 94.153,Z 65.067,A 180.000,B 0.000,C 180.000} C_DIS
LIN {X 48.281,Y 94.218,Z 65.065,A 180.000,B 0.000,C 180.000} C_DIS
LIN {X 48.015,Y 94.609,Z 65.048,A 180.000,B 0.000,C 180.000} C_DIS
LIN {X 47.971,Y 94.674,Z 65.045,A 180.000,B 0.000,C 180.000} C_DIS
LIN {X 47.927,Y 94.740,Z 65.043,A 180.000,B 0.000,C 180.000} C_DIS
LIN {X 47.885,Y 94.806,Z 65.040,A 180.000,B 0.000,C 180.000} C_DIS
LIN {X 47.844,Y 94.874,Z 65.037,A 180.000,B 0.000,C 180.000} C_DIS
LIN {X 47.564,Y 95.348,Z 65.018,A 180.000,B 0.000,C 180.000} C_DIS
LIN {X 47.524,Y 95.416,Z 65.015,A 180.000,B 0.000,C 180.000} C_DIS
LIN {X 47.486,Y 95.485,Z 65.012,A 180.000,B 0.000,C 180.000} C_DIS
LIN {X 47.450,Y 95.555,Z 65.010,A 180.000,B 0.000,C 180.000} C_DIS
LIN {X 47.199,Y 96.046,Z 64.990,A 180.000,B 0.000,C 180.000} C_DIS
LIN {X 47.164,Y 96.116,Z 64.988,A 180.000,B 0.000,C 180.000} C_DIS
LIN {X 47.130,Y 96.188,Z 64.985,A 180.000,B 0.000,C 180.000} C_DIS
LIN {X 47.098,Y 96.260,Z 64.982,A 180.000,B 0.000,C 180.000} C_DIS
LIN {X 46.879,Y 96.766,Z 64.963,A 180.000,B 0.000,C 180.000} C_DIS
LIN {X 46.848,Y 96.838,Z 64.960,A 180.000,B 0.000,C 180.000} C_DIS
LIN {X 46.819,Y 96.911,Z 64.957,A 180.000,B 0.000,C 180.000} C_DIS
LIN {X 46.792,Y 96.985,Z 64.955,A 180.000,B 0.000,C 180.000} C_DIS
LIN {X 46.605,Y 97.504,Z 64.935,A 180.000,B 0.000,C 180.000} C_DIS
LIN {X 46.579,Y 97.578,Z 64.933,A 180.000,B 0.000,C 180.000} C_DIS
LIN {X 46.554,Y 97.653,Z 64.930,A 180.000,B 0.000,C 180.000} C_DIS
LIN {X 46.532,Y 97.728,Z 64.927,A 180.000,B 0.000,C 180.000} C_DIS
LIN {X 46.378,Y 98.258,Z 64.908,A 180.000,B 0.000,C 180.000} C_DIS
LIN {X 46.356,Y 98.333,Z 64.905,A 180.000,B 0.000,C 180.000} C_DIS
LIN {X 46.337,Y 98.410,Z 64.902,A 180.000,B 0.000,C 180.000} C_DIS
LIN {X 46.319,Y 98.486,Z 64.900,A 180.000,B 0.000,C 180.000} C_DIS
LIN {X 46.267,Y 98.717,Z 64.891,A 180.000,B 0.000,C 180.000} C_DIS
LIN {X 46.233,Y 98.871,Z 64.886,A 180.000,B 0.000,C 180.000} C_DIS
LIN {X 46.199,Y 99.024,Z 64.880,A 180.000,B 0.000,C 180.000} C_DIS
LIN {X 46.182,Y 99.101,Z 64.878,A 180.000,B 0.000,C 180.000} C_DIS
LIN {X 46.167,Y 99.178,Z 64.875,A 180.000,B 0.000,C 180.000} C_DIS
LIN {X 46.154,Y 99.256,Z 64.872,A 180.000,B 0.000,C 180.000} C_DIS
LIN {X 46.068,Y 99.801,Z 64.853,A 180.000,B 0.000,C 180.000} C_DIS
LIN {X 46.056,Y 99.878,Z 64.850,A 180.000,B 0.000,C 180.000} C_DIS
LIN {X 46.045,Y 99.957,Z 64.847,A 180.000,B 0.000,C 180.000} C_DIS
LIN {X 46.038,Y 100.035,Z 64.845,A 180.000,B 0.000,C 180.000} C_DIS
LIN {X 46.015,Y 100.270,Z 64.836,A 180.000,B 0.000,C 180.000} C_DIS
LIN {X 46.008,Y 100.349,Z 64.834,A 180.000,B 0.000,C 180.000} C_DIS
LIN {X 45.993,Y 100.505,Z 64.828,A 180.000,B 0.000,C 180.000} C_DIS
LIN {X 45.986,Y 100.584,Z 64.825,A 180.000,B 0.000,C 180.000} C_DIS
LIN {X 45.978,Y 100.662,Z 64.823,A 180.000,B 0.000,C 180.000} C_DIS
LIN {X 45.973,Y 100.741,Z 64.820,A 180.000,B 0.000,C 180.000} C_DIS
LIN {X 45.970,Y 100.819,Z 64.817,A 180.000,B 0.000,C 180.000} C_DIS
LIN {X 45.955,Y 101.292,Z 64.801,A 180.000,B 0.000,C 180.000} C_DIS
LIN {X 45.953,Y 101.370,Z 64.798,A 180.000,B 0.000,C 180.000} C_DIS
LIN {X 45.951,Y 101.449,Z 64.795,A 180.000,B 0.000,C 180.000} C_DIS
LIN {X 45.950,Y 101.528,Z 64.792,A 180.000,B 0.000,C 180.000} C_DIS
LIN {X 45.952,Y 101.607,Z 64.790,A 180.000,B 0.000,C 180.000} C_DIS
LIN {X 45.957,Y 101.764,Z 64.784,A 180.000,B 0.000,C 180.000} C_DIS
LIN {X 45.964,Y 102.000,Z 64.776,A 180.000,B 0.000,C 180.000} C_DIS
LIN {X 45.969,Y 102.158,Z 64.770,A 180.000,B 0.000,C 180.000} C_DIS
LIN {X 45.972,Y 102.236,Z 64.768,A 180.000,B 0.000,C 180.000} C_DIS
LIN {X 45.977,Y 102.315,Z 64.765,A 180.000,B 0.000,C 180.000} C_DIS
LIN {X 45.983,Y 102.393,Z 64.762,A 180.000,B 0.000,C 180.000} C_DIS
LIN {X 46.006,Y 102.629,Z 64.754,A 180.000,B 0.000,C 180.000} C_DIS
LIN {X 46.021,Y 102.785,Z 64.748,A 180.000,B 0.000,C 180.000} C_DIS
LIN {X 46.028,Y 102.864,Z 64.746,A 180.000,B 0.000,C 180.000} C_DIS
LIN {X 46.035,Y 102.942,Z 64.743,A 180.000,B 0.000,C 180.000} C_DIS
LIN {X 46.043,Y 103.021,Z 64.740,A 180.000,B 0.000,C 180.000} C_DIS
LIN {X 46.052,Y 103.099,Z 64.737,A 180.000,B 0.000,C 180.000} C_DIS
LIN {X 46.064,Y 103.177,Z 64.735,A 180.000,B 0.000,C 180.000} C_DIS
LIN {X 46.089,Y 103.332,Z 64.729,A 180.000,B 0.000,C 180.000} C_DIS
LIN {X 46.126,Y 103.566,Z 64.721,A 180.000,B 0.000,C 180.000} C_DIS
LIN {X 46.150,Y 103.721,Z 64.715,A 180.000,B 0.000,C 180.000} C_DIS
LIN {X 46.163,Y 103.799,Z 64.713,A 180.000,B 0.000,C 180.000} C_DIS
LIN {X 46.177,Y 103.876,Z 64.710,A 180.000,B 0.000,C 180.000} C_DIS
LIN {X 46.194,Y 103.953,Z 64.707,A 180.000,B 0.000,C 180.000} C_DIS
LIN {X 46.245,Y 104.184,Z 64.699,A 180.000,B 0.000,C 180.000} C_DIS
LIN {X 46.280,Y 104.338,Z 64.693,A 180.000,B 0.000,C 180.000} C_DIS
LIN {X 46.314,Y 104.491,Z 64.688,A 180.000,B 0.000,C 180.000} C_DIS
LIN {X 46.331,Y 104.568,Z 64.685,A 180.000,B 0.000,C 180.000} C_DIS
LIN {X 46.350,Y 104.644,Z 64.682,A 180.000,B 0.000,C 180.000} C_DIS
LIN {X 46.372,Y 104.720,Z 64.680,A 180.000,B 0.000,C 180.000} C_DIS
LIN {X 46.416,Y 104.872,Z 64.674,A 180.000,B 0.000,C 180.000} C_DIS
LIN {X 46.460,Y 105.023,Z 64.669,A 180.000,B 0.000,C 180.000} C_DIS
LIN {X 46.504,Y 105.174,Z 64.664,A 180.000,B 0.000,C 180.000} C_DIS
LIN {X 46.526,Y 105.250,Z 64.661,A 180.000,B 0.000,C 180.000} C_DIS
LIN {X 46.548,Y 105.325,Z 64.659,A 180.000,B 0.000,C 180.000} C_DIS
LIN {X 46.572,Y 105.400,Z 64.656,A 180.000,B 0.000,C 180.000} C_DIS
LIN {X 46.598,Y 105.475,Z 64.654,A 180.000,B 0.000,C 180.000} C_DIS
LIN {X 46.624,Y 105.549,Z 64.651,A 180.000,B 0.000,C 180.000} C_DIS
LIN {X 46.651,Y 105.623,Z 64.649,A 180.000,B 0.000,C 180.000} C_DIS
LIN {X 46.704,Y 105.771,Z 64.644,A 180.000,B 0.000,C 180.000} C_DIS
LIN {X 46.758,Y 105.919,Z 64.639,A 180.000,B 0.000,C 180.000} C_DIS
LIN {X 46.811,Y 106.067,Z 64.634,A 180.000,B 0.000,C 180.000} C_DIS
LIN {X 46.870,Y 106.213,Z 64.629,A 180.000,B 0.000,C 180.000} C_DIS
LIN {X 46.933,Y 106.358,Z 64.624,A 180.000,B 0.000,C 180.000} C_DIS
LIN {X 46.995,Y 106.502,Z 64.620,A 180.000,B 0.000,C 180.000} C_DIS
LIN {X 47.058,Y 106.647,Z 64.615,A 180.000,B 0.000,C 180.000} C_DIS
LIN {X 47.121,Y 106.791,Z 64.610,A 180.000,B 0.000,C 180.000} C_DIS
LIN {X 47.189,Y 106.933,Z 64.606,A 180.000,B 0.000,C 180.000} C_DIS
LIN {X 47.260,Y 107.074,Z 64.602,A 180.000,B 0.000,C 180.000} C_DIS
LIN {X 47.332,Y 107.214,Z 64.597,A 180.000,B 0.000,C 180.000} C_DIS
LIN {X 47.403,Y 107.354,Z 64.593,A 180.000,B 0.000,C 180.000} C_DIS
LIN {X 47.475,Y 107.495,Z 64.589,A 180.000,B 0.000,C 180.000} C_DIS
LIN {X 47.552,Y 107.632,Z 64.585,A 180.000,B 0.000,C 180.000} C_DIS
LIN {X 47.632,Y 107.768,Z 64.581,A 180.000,B 0.000,C 180.000} C_DIS
LIN {X 47.712,Y 107.903,Z 64.577,A 180.000,B 0.000,C 180.000} C_DIS
LIN {X 47.792,Y 108.039,Z 64.573,A 180.000,B 0.000,C 180.000} C_DIS
LIN {X 47.873,Y 108.174,Z 64.570,A 180.000,B 0.000,C 180.000} C_DIS
LIN {X 47.958,Y 108.307,Z 64.566,A 180.000,B 0.000,C 180.000} C_DIS
LIN {X 48.047,Y 108.437,Z 64.562,A 180.000,B 0.000,C 180.000} C_DIS
LIN {X 48.135,Y 108.567,Z 64.559,A 180.000,B 0.000,C 180.000} C_DIS
LIN {X 48.224,Y 108.698,Z 64.556,A 180.000,B 0.000,C 180.000} C_DIS
LIN {X 48.312,Y 108.828,Z 64.552,A 180.000,B 0.000,C 180.000} C_DIS
LIN {X 48.406,Y 108.954,Z 64.549,A 180.000,B 0.000,C 180.000} C_DIS
LIN {X 48.502,Y 109.079,Z 64.546,A 180.000,B 0.000,C 180.000} C_DIS
LIN {X 48.599,Y 109.203,Z 64.543,A 180.000,B 0.000,C 180.000} C_DIS
LIN {X 48.695,Y 109.328,Z 64.540,A 180.000,B 0.000,C 180.000} C_DIS
LIN {X 48.792,Y 109.452,Z 64.537,A 180.000,B 0.000,C 180.000} C_DIS
LIN {X 48.893,Y 109.573,Z 64.534,A 180.000,B 0.000,C 180.000} C_DIS
LIN {X 48.997,Y 109.691,Z 64.532,A 180.000,B 0.000,C 180.000} C_DIS
LIN {X 49.101,Y 109.809,Z 64.529,A 180.000,B 0.000,C 180.000} C_DIS
LIN {X 49.205,Y 109.927,Z 64.527,A 180.000,B 0.000,C 180.000} C_DIS
LIN {X 49.418,Y 110.160,Z 64.522,A 180.000,B 0.000,C 180.000} C_DIS
LIN {X 49.641,Y 110.382,Z 64.518,A 180.000,B 0.000,C 180.000} C_DIS
LIN {X 49.864,Y 110.605,Z 64.514,A 180.000,B 0.000,C 180.000} C_DIS
LIN {X 50.097,Y 110.816,Z 64.511,A 180.000,B 0.000,C 180.000} C_DIS
LIN {X 50.334,Y 111.025,Z 64.508,A 180.000,B 0.000,C 180.000} C_DIS
LIN {X 50.574,Y 111.228,Z 64.505,A 180.000,B 0.000,C 180.000} C_DIS
LIN {X 50.823,Y 111.421,Z 64.503,A 180.000,B 0.000,C 180.000} C_DIS
LIN {X 51.072,Y 111.615,Z 64.502,A 180.000,B 0.000,C 180.000} C_DIS
LIN {X 51.330,Y 111.795,Z 64.501,A 180.000,B 0.000,C 180.000} C_DIS
LIN {X 51.590,Y 111.972,Z 64.500,A 180.000,B 0.000,C 180.000} C_DIS
LIN {X 51.783,Y 112.101,Z 64.500,A 180.000,B 0.000,C 180.000} C_DIS
; Cutting Move Starts
LIN {X 51.847,Y 112.140,Z 64.500,A 180.000,B 0.000,C 180.000} C_DIS
LIN {X 52.383,Y 112.457,Z 64.500,A 180.000,B 0.000,C 180.000} C_DIS
LIN {X 52.562,Y 112.554,Z 64.500,A 180.000,B 0.000,C 180.000} C_DIS
LIN {X 53.059,Y 112.807,Z 64.500,A 180.000,B 0.000,C 180.000} C_DIS
LIN {X 53.098,Y 112.827,Z 64.500,A 180.000,B 0.000,C 180.000} C_DIS
LIN {X 53.277,Y 112.909,Z 64.500,A 180.000,B 0.000,C 180.000} C_DIS
LIN {X 53.813,Y 113.141,Z 64.500,A 180.000,B 0.000,C 180.000} C_DIS
LIN {X 53.870,Y 113.165,Z 64.500,A 180.000,B 0.000,C 180.000} C_DIS
LIN {X 53.992,Y 113.210,Z 64.500,A 180.000,B 0.000,C 180.000} C_DIS
LIN {X 54.528,Y 113.403,Z 64.500,A 180.000,B 0.000,C 180.000} C_DIS
LIN {X 54.707,Y 113.462,Z 64.500,A 180.000,B 0.000,C 180.000} C_DIS
LIN {X 55.243,Y 113.618,Z 64.500,A 180.000,B 0.000,C 180.000} C_DIS
LIN {X 55.422,Y 113.666,Z 64.500,A 180.000,B 0.000,C 180.000} C_DIS
LIN {X 55.575,Y 113.701,Z 64.500,A 180.000,B 0.000,C 180.000} C_DIS
LIN {X 55.958,Y 113.786,Z 64.500,A 180.000,B 0.000,C 180.000} C_DIS
LIN {X 56.137,Y 113.826,Z 64.500,A 180.000,B 0.000,C 180.000} C_DIS
LIN {X 56.316,Y 113.855,Z 64.500,A 180.000,B 0.000,C 180.000} C_DIS
LIN {X 56.852,Y 113.940,Z 64.500,A 180.000,B 0.000,C 180.000} C_DIS
LIN {X 57.031,Y 113.962,Z 64.500,A 180.000,B 0.000,C 180.000} C_DIS
LIN {X 57.567,Y 114.013,Z 64.500,A 180.000,B 0.000,C 180.000} C_DIS
LIN {X 57.746,Y 114.027,Z 64.500,A 180.000,B 0.000,C 180.000} C_DIS
LIN {X 57.925,Y 114.033,Z 64.500,A 180.000,B 0.000,C 180.000} C_DIS
LIN {X 58.282,Y 114.044,Z 64.500,A 180.000,B 0.000,C 180.000} C_DIS
LIN {X 58.461,Y 114.050,Z 64.500,A 180.000,B 0.000,C 180.000} C_DIS
LIN {X 58.640,Y 114.047,Z 64.500,A 180.000,B 0.000,C 180.000} C_DIS
LIN {X 59.176,Y 114.030,Z 64.500,A 180.000,B 0.000,C 180.000} C_DIS
LIN {X 59.355,Y 114.020,Z 64.500,A 180.000,B 0.000,C 180.000} C_DIS
LIN {X 59.534,Y 114.003,Z 64.500,A 180.000,B 0.000,C 180.000} C_DIS
LIN {X 59.891,Y 113.969,Z 64.500,A 180.000,B 0.000,C 180.000} C_DIS
LIN {X 60.070,Y 113.951,Z 64.500,A 180.000,B 0.000,C 180.000} C_DIS
LIN {X 60.249,Y 113.924,Z 64.500,A 180.000,B 0.000,C 180.000} C_DIS
LIN {X 60.606,Y 113.868,Z 64.500,A 180.000,B 0.000,C 180.000} C_DIS
LIN {X 60.785,Y 113.839,Z 64.500,A 180.000,B 0.000,C 180.000} C_DIS
LIN {X 60.964,Y 113.804,Z 64.500,A 180.000,B 0.000,C 180.000} C_DIS
LIN {X 61.500,Y 113.684,Z 64.500,A 180.000,B 0.000,C 180.000} C_DIS
LIN {X 61.679,Y 113.640,Z 64.500,A 180.000,B 0.000,C 180.000} C_DIS
LIN {X 61.858,Y 113.588,Z 64.500,A 180.000,B 0.000,C 180.000} C_DIS
LIN {X 62.215,Y 113.484,Z 64.500,A 180.000,B 0.000,C 180.000} C_DIS
LIN {X 62.394,Y 113.431,Z 64.500,A 180.000,B 0.000,C 180.000} C_DIS
LIN {X 62.573,Y 113.367,Z 64.500,A 180.000,B 0.000,C 180.000} C_DIS
LIN {X 62.930,Y 113.238,Z 64.500,A 180.000,B 0.000,C 180.000} C_DIS
LIN {X 63.109,Y 113.173,Z 64.500,A 180.000,B 0.000,C 180.000} C_DIS
LIN {X 63.130,Y 113.165,Z 64.500,A 180.000,B 0.000,C 180.000} C_DIS
LIN {X 63.288,Y 113.097,Z 64.500,A 180.000,B 0.000,C 180.000} C_DIS
LIN {X 63.645,Y 112.943,Z 64.500,A 180.000,B 0.000,C 180.000} C_DIS
LIN {X 63.824,Y 112.865,Z 64.500,A 180.000,B 0.000,C 180.000} C_DIS
LIN {X 63.941,Y 112.807,Z 64.500,A 180.000,B 0.000,C 180.000} C_DIS
LIN {X 64.360,Y 112.594,Z 64.500,A 180.000,B 0.000,C 180.000} C_DIS
LIN {X 64.539,Y 112.501,Z 64.500,A 180.000,B 0.000,C 180.000} C_DIS
LIN {X 64.630,Y 112.450,Z 64.500,A 180.000,B 0.000,C 180.000} C_DIS
LIN {X 65.075,Y 112.186,Z 64.500,A 180.000,B 0.000,C 180.000} C_DIS
LIN {X 65.231,Y 112.092,Z 64.500,A 180.000,B 0.000,C 180.000} C_DIS
LIN {X 65.254,Y 112.077,Z 64.500,A 180.000,B 0.000,C 180.000} C_DIS
LIN {X 65.433,Y 111.956,Z 64.500,A 180.000,B 0.000,C 180.000} C_DIS
LIN {X 65.791,Y 111.713,Z 64.500,A 180.000,B 0.000,C 180.000} C_DIS
LIN {X 65.969,Y 111.583,Z 64.500,A 180.000,B 0.000,C 180.000} C_DIS
LIN {X 66.327,Y 111.306,Z 64.500,A 180.000,B 0.000,C 180.000} C_DIS
LIN {X 66.465,Y 111.198,Z 64.500,A 180.000,B 0.000,C 180.000} C_DIS
LIN {X 66.506,Y 111.165,Z 64.500,A 180.000,B 0.000,C 180.000} C_DIS
LIN {X 66.672,Y 111.019,Z 64.500,A 180.000,B 0.000,C 180.000} C_DIS
LIN {X 66.875,Y 110.841,Z 64.500,A 180.000,B 0.000,C 180.000} C_DIS
LIN {X 67.042,Y 110.693,Z 64.500,A 180.000,B 0.000,C 180.000} C_DIS
LIN {X 67.077,Y 110.662,Z 64.500,A 180.000,B 0.000,C 180.000} C_DIS
LIN {X 67.221,Y 110.521,Z 64.500,A 180.000,B 0.000,C 180.000} C_DIS
LIN {X 67.578,Y 110.163,Z 64.500,A 180.000,B 0.000,C 180.000} C_DIS
LIN {X 67.616,Y 110.126,Z 64.500,A 180.000,B 0.000,C 180.000} C_DIS
LIN {X 67.757,Y 109.970,Z 64.500,A 180.000,B 0.000,C 180.000} C_DIS
LIN {X 68.115,Y 109.564,Z 64.500,A 180.000,B 0.000,C 180.000} C_DIS
LIN {X 68.241,Y 109.410,Z 64.500,A 180.000,B 0.000,C 180.000} C_DIS
LIN {X 68.518,Y 109.053,Z 64.500,A 180.000,B 0.000,C 180.000} C_DIS
LIN {X 68.651,Y 108.880,Z 64.500,A 180.000,B 0.000,C 180.000} C_DIS
LIN {X 68.655,Y 108.874,Z 64.500,A 180.000,B 0.000,C 180.000} C_DIS
LIN {X 68.778,Y 108.695,Z 64.500,A 180.000,B 0.000,C 180.000} C_DIS
LIN {X 69.021,Y 108.338,Z 64.500,A 180.000,B 0.000,C 180.000} C_DIS
LIN {X 69.137,Y 108.159,Z 64.500,A 180.000,B 0.000,C 180.000} C_DIS
LIN {X 69.454,Y 107.623,Z 64.500,A 180.000,B 0.000,C 180.000} C_DIS
LIN {X 69.545,Y 107.456,Z 64.500,A 180.000,B 0.000,C 180.000} C_DIS
LIN {X 69.733,Y 107.086,Z 64.500,A 180.000,B 0.000,C 180.000} C_DIS
LIN {X 69.824,Y 106.908,Z 64.500,A 180.000,B 0.000,C 180.000} C_DIS
LIN {X 69.902,Y 106.739,Z 64.500,A 180.000,B 0.000,C 180.000} C_DIS
LIN {X 70.139,Y 106.193,Z 64.500,A 180.000,B 0.000,C 180.000} C_DIS
LIN {X 70.208,Y 106.014,Z 64.500,A 180.000,B 0.000,C 180.000} C_DIS
LIN {X 70.401,Y 105.477,Z 64.500,A 180.000,B 0.000,C 180.000} C_DIS
LIN {X 70.439,Y 105.369,Z 64.500,A 180.000,B 0.000,C 180.000} C_DIS
LIN {X 70.460,Y 105.299,Z 64.500,A 180.000,B 0.000,C 180.000} C_DIS
LIN {X 70.617,Y 104.758,Z 64.500,A 180.000,B 0.000,C 180.000} C_DIS
LIN {X 70.665,Y 104.584,Z 64.500,A 180.000,B 0.000,C 180.000} C_DIS
LIN {X 70.705,Y 104.405,Z 64.500,A 180.000,B 0.000,C 180.000} C_DIS
LIN {X 70.796,Y 103.999,Z 64.500,A 180.000,B 0.000,C 180.000} C_DIS
LIN {X 70.824,Y 103.869,Z 64.500,A 180.000,B 0.000,C 180.000} C_DIS
LIN {X 70.855,Y 103.690,Z 64.500,A 180.000,B 0.000,C 180.000} C_DIS
LIN {X 70.940,Y 103.153,Z 64.500,A 180.000,B 0.000,C 180.000} C_DIS
LIN {X 70.962,Y 102.975,Z 64.500,A 180.000,B 0.000,C 180.000} C_DIS
LIN {X 71.012,Y 102.438,Z 64.500,A 180.000,B 0.000,C 180.000} C_DIS
LIN {X 71.027,Y 102.260,Z 64.500,A 180.000,B 0.000,C 180.000} C_DIS
LIN {X 71.033,Y 102.081,Z 64.500,A 180.000,B 0.000,C 180.000} C_DIS
LIN {X 71.044,Y 101.723,Z 64.500,A 180.000,B 0.000,C 180.000} C_DIS
LIN {X 71.050,Y 101.545,Z 64.500,A 180.000,B 0.000,C 180.000} C_DIS
LIN {X 71.047,Y 101.366,Z 64.500,A 180.000,B 0.000,C 180.000} C_DIS
LIN {X 71.030,Y 100.829,Z 64.500,A 180.000,B 0.000,C 180.000} C_DIS
LIN {X 71.021,Y 100.651,Z 64.500,A 180.000,B 0.000,C 180.000} C_DIS
LIN {X 71.004,Y 100.472,Z 64.500,A 180.000,B 0.000,C 180.000} C_DIS
LIN {X 70.970,Y 100.114,Z 64.500,A 180.000,B 0.000,C 180.000} C_DIS
LIN {X 70.952,Y 99.936,Z 64.500,A 180.000,B 0.000,C 180.000} C_DIS
LIN {X 70.925,Y 99.757,Z 64.500,A 180.000,B 0.000,C 180.000} C_DIS
LIN {X 70.840,Y 99.221,Z 64.500,A 180.000,B 0.000,C 180.000} C_DIS
LIN {X 70.805,Y 99.042,Z 64.500,A 180.000,B 0.000,C 180.000} C_DIS
LIN {X 70.718,Y 98.654,Z 64.500,A 180.000,B 0.000,C 180.000} C_DIS
LIN {X 70.685,Y 98.505,Z 64.500,A 180.000,B 0.000,C 180.000} C_DIS
LIN {X 70.642,Y 98.327,Z 64.500,A 180.000,B 0.000,C 180.000} C_DIS
LIN {X 70.617,Y 98.242,Z 64.500,A 180.000,B 0.000,C 180.000} C_DIS
LIN {X 70.486,Y 97.790,Z 64.500,A 180.000,B 0.000,C 180.000} C_DIS
LIN {X 70.439,Y 97.631,Z 64.500,A 180.000,B 0.000,C 180.000} C_DIS
LIN {X 70.432,Y 97.612,Z 64.500,A 180.000,B 0.000,C 180.000} C_DIS
LIN {X 70.369,Y 97.433,Z 64.500,A 180.000,B 0.000,C 180.000} C_DIS
LIN {X 70.240,Y 97.075,Z 64.500,A 180.000,B 0.000,C 180.000} C_DIS
LIN {X 70.175,Y 96.897,Z 64.500,A 180.000,B 0.000,C 180.000} C_DIS
LIN {X 70.100,Y 96.718,Z 64.500,A 180.000,B 0.000,C 180.000} C_DIS
LIN {X 69.902,Y 96.261,Z 64.500,A 180.000,B 0.000,C 180.000} C_DIS
LIN {X 69.867,Y 96.181,Z 64.500,A 180.000,B 0.000,C 180.000} C_DIS
LIN {X 69.779,Y 96.003,Z 64.500,A 180.000,B 0.000,C 180.000} C_DIS
LIN {X 69.545,Y 95.544,Z 64.500,A 180.000,B 0.000,C 180.000} C_DIS
LIN {X 69.504,Y 95.466,Z 64.500,A 180.000,B 0.000,C 180.000} C_DIS
LIN {X 69.401,Y 95.288,Z 64.500,A 180.000,B 0.000,C 180.000} C_DIS
LIN {X 69.187,Y 94.927,Z 64.500,A 180.000,B 0.000,C 180.000} C_DIS
LIN {X 69.081,Y 94.751,Z 64.500,A 180.000,B 0.000,C 180.000} C_DIS
LIN {X 69.008,Y 94.644,Z 64.500,A 180.000,B 0.000,C 180.000} C_DIS
LIN {X 68.717,Y 94.215,Z 64.500,A 180.000,B 0.000,C 180.000} C_DIS
LIN {X 68.651,Y 94.120,Z 64.500,A 180.000,B 0.000,C 180.000} C_DIS
LIN {X 68.587,Y 94.036,Z 64.500,A 180.000,B 0.000,C 180.000} C_DIS
LIN {X 68.293,Y 93.657,Z 64.500,A 180.000,B 0.000,C 180.000} C_DIS
LIN {X 68.170,Y 93.500,Z 64.500,A 180.000,B 0.000,C 180.000} C_DIS
LIN {X 68.115,Y 93.436,Z 64.500,A 180.000,B 0.000,C 180.000} C_DIS
LIN {X 67.698,Y 92.964,Z 64.500,A 180.000,B 0.000,C 180.000} C_DIS
LIN {X 67.578,Y 92.837,Z 64.500,A 180.000,B 0.000,C 180.000} C_DIS
LIN {X 67.169,Y 92.427,Z 64.500,A 180.000,B 0.000,C 180.000} C_DIS
LIN {X 67.042,Y 92.307,Z 64.500,A 180.000,B 0.000,C 180.000} C_DIS
LIN {X 66.976,Y 92.249,Z 64.500,A 180.000,B 0.000,C 180.000} C_DIS
LIN {X 66.571,Y 91.891,Z 64.500,A 180.000,B 0.000,C 180.000} C_DIS
LIN {X 66.506,Y 91.835,Z 64.500,A 180.000,B 0.000,C 180.000} C_DIS
LIN {X 66.350,Y 91.712,Z 64.500,A 180.000,B 0.000,C 180.000} C_DIS
LIN {X 65.969,Y 91.417,Z 64.500,A 180.000,B 0.000,C 180.000} C_DIS
LIN {X 65.887,Y 91.355,Z 64.500,A 180.000,B 0.000,C 180.000} C_DIS
LIN {X 65.791,Y 91.287,Z 64.500,A 180.000,B 0.000,C 180.000} C_DIS
LIN {X 65.364,Y 90.997,Z 64.500,A 180.000,B 0.000,C 180.000} C_DIS
LIN {X 65.254,Y 90.923,Z 64.500,A 180.000,B 0.000,C 180.000} C_DIS
LIN {X 65.083,Y 90.818,Z 64.500,A 180.000,B 0.000,C 180.000} C_DIS
LIN {X 64.718,Y 90.603,Z 64.500,A 180.000,B 0.000,C 180.000} C_DIS
LIN {X 64.539,Y 90.499,Z 64.500,A 180.000,B 0.000,C 180.000} C_DIS
LIN {X 64.467,Y 90.461,Z 64.500,A 180.000,B 0.000,C 180.000} C_DIS
LIN {X 64.003,Y 90.224,Z 64.500,A 180.000,B 0.000,C 180.000} C_DIS
LIN {X 63.824,Y 90.135,Z 64.500,A 180.000,B 0.000,C 180.000} C_DIS
LIN {X 63.752,Y 90.103,Z 64.500,A 180.000,B 0.000,C 180.000} C_DIS
LIN {X 63.288,Y 89.903,Z 64.500,A 180.000,B 0.000,C 180.000} C_DIS
LIN {X 63.141,Y 89.840,Z 64.500,A 180.000,B 0.000,C 180.000} C_DIS
LIN {X 63.109,Y 89.827,Z 64.500,A 180.000,B 0.000,C 180.000} C_DIS
LIN {X 62.930,Y 89.762,Z 64.500,A 180.000,B 0.000,C 180.000} C_DIS
LIN {X 62.573,Y 89.633,Z 64.500,A 180.000,B 0.000,C 180.000} C_DIS
LIN {X 62.394,Y 89.569,Z 64.500,A 180.000,B 0.000,C 180.000} C_DIS
LIN {X 62.387,Y 89.567,Z 64.500,A 180.000,B 0.000,C 180.000} C_DIS
LIN {X 62.215,Y 89.516,Z 64.500,A 180.000,B 0.000,C 180.000} C_DIS
LIN {X 61.777,Y 89.388,Z 64.500,A 180.000,B 0.000,C 180.000} C_DIS
LIN {X 61.679,Y 89.360,Z 64.500,A 180.000,B 0.000,C 180.000} C_DIS
LIN {X 61.500,Y 89.316,Z 64.500,A 180.000,B 0.000,C 180.000} C_DIS
LIN {X 60.964,Y 89.196,Z 64.500,A 180.000,B 0.000,C 180.000} C_DIS
LIN {X 60.785,Y 89.161,Z 64.500,A 180.000,B 0.000,C 180.000} C_DIS
LIN {X 60.606,Y 89.132,Z 64.500,A 180.000,B 0.000,C 180.000} C_DIS
LIN {X 60.249,Y 89.076,Z 64.500,A 180.000,B 0.000,C 180.000} C_DIS
LIN {X 60.070,Y 89.049,Z 64.500,A 180.000,B 0.000,C 180.000} C_DIS
LIN {X 59.892,Y 89.031,Z 64.500,A 180.000,B 0.000,C 180.000} C_DIS
LIN {X 59.534,Y 88.997,Z 64.500,A 180.000,B 0.000,C 180.000} C_DIS
LIN {X 59.355,Y 88.980,Z 64.500,A 180.000,B 0.000,C 180.000} C_DIS
LIN {X 59.176,Y 88.970,Z 64.500,A 180.000,B 0.000,C 180.000} C_DIS
LIN {X 58.640,Y 88.953,Z 64.500,A 180.000,B 0.000,C 180.000} C_DIS
LIN {X 58.461,Y 88.950,Z 64.500,A 180.000,B 0.000,C 180.000} C_DIS
LIN {X 58.282,Y 88.956,Z 64.500,A 180.000,B 0.000,C 180.000} C_DIS
LIN {X 57.925,Y 88.967,Z 64.500,A 180.000,B 0.000,C 180.000} C_DIS
LIN {X 57.746,Y 88.973,Z 64.500,A 180.000,B 0.000,C 180.000} C_DIS
LIN {X 57.567,Y 88.987,Z 64.500,A 180.000,B 0.000,C 180.000} C_DIS
LIN {X 57.031,Y 89.038,Z 64.500,A 180.000,B 0.000,C 180.000} C_DIS
LIN {X 56.852,Y 89.060,Z 64.500,A 180.000,B 0.000,C 180.000} C_DIS
LIN {X 56.316,Y 89.145,Z 64.500,A 180.000,B 0.000,C 180.000} C_DIS
LIN {X 56.137,Y 89.174,Z 64.500,A 180.000,B 0.000,C 180.000} C_DIS
LIN {X 55.977,Y 89.209,Z 64.500,A 180.000,B 0.000,C 180.000} C_DIS
LIN {X 55.601,Y 89.293,Z 64.500,A 180.000,B 0.000,C 180.000} C_DIS
LIN {X 55.422,Y 89.334,Z 64.500,A 180.000,B 0.000,C 180.000} C_DIS
LIN {X 55.243,Y 89.382,Z 64.500,A 180.000,B 0.000,C 180.000} C_DIS
LIN {X 54.707,Y 89.538,Z 64.500,A 180.000,B 0.000,C 180.000} C_DIS
LIN {X 54.613,Y 89.567,Z 64.500,A 180.000,B 0.000,C 180.000} C_DIS
LIN {X 54.528,Y 89.597,Z 64.500,A 180.000,B 0.000,C 180.000} C_DIS
LIN {X 53.992,Y 89.790,Z 64.500,A 180.000,B 0.000,C 180.000} C_DIS
LIN {X 53.813,Y 89.859,Z 64.500,A 180.000,B 0.000,C 180.000} C_DIS
LIN {X 53.455,Y 90.014,Z 64.500,A 180.000,B 0.000,C 180.000} C_DIS
LIN {X 53.248,Y 90.103,Z 64.500,A 180.000,B 0.000,C 180.000} C_DIS
LIN {X 53.098,Y 90.173,Z 64.500,A 180.000,B 0.000,C 180.000} C_DIS
LIN {X 52.919,Y 90.264,Z 64.500,A 180.000,B 0.000,C 180.000} C_DIS
LIN {X 52.533,Y 90.461,Z 64.500,A 180.000,B 0.000,C 180.000} C_DIS
LIN {X 52.383,Y 90.543,Z 64.500,A 180.000,B 0.000,C 180.000} C_DIS
LIN {X 51.847,Y 90.860,Z 64.500,A 180.000,B 0.000,C 180.000} C_DIS
LIN {X 51.668,Y 90.975,Z 64.500,A 180.000,B 0.000,C 180.000} C_DIS
LIN {X 51.310,Y 91.218,Z 64.500,A 180.000,B 0.000,C 180.000} C_DIS
LIN {X 51.131,Y 91.341,Z 64.500,A 180.000,B 0.000,C 180.000} C_DIS
LIN {X 51.113,Y 91.355,Z 64.500,A 180.000,B 0.000,C 180.000} C_DIS
LIN {X 50.953,Y 91.478,Z 64.500,A 180.000,B 0.000,C 180.000} C_DIS
LIN {X 50.595,Y 91.755,Z 64.500,A 180.000,B 0.000,C 180.000} C_DIS
LIN {X 50.429,Y 91.891,Z 64.500,A 180.000,B 0.000,C 180.000} C_DIS
LIN {X 50.024,Y 92.249,Z 64.500,A 180.000,B 0.000,C 180.000} C_DIS
LIN {X 49.880,Y 92.379,Z 64.500,A 180.000,B 0.000,C 180.000} C_DIS
LIN {X 49.831,Y 92.427,Z 64.500,A 180.000,B 0.000,C 180.000} C_DIS
LIN {X 49.474,Y 92.785,Z 64.500,A 180.000,B 0.000,C 180.000} C_DIS
LIN {X 49.344,Y 92.917,Z 64.500,A 180.000,B 0.000,C 180.000} C_DIS
LIN {X 49.302,Y 92.964,Z 64.500,A 180.000,B 0.000,C 180.000} C_DIS
LIN {X 48.986,Y 93.321,Z 64.500,A 180.000,B 0.000,C 180.000} C_DIS
LIN {X 48.830,Y 93.500,Z 64.500,A 180.000,B 0.000,C 180.000} C_DIS
LIN {X 48.807,Y 93.528,Z 64.500,A 180.000,B 0.000,C 180.000} C_DIS
LIN {X 48.690,Y 93.679,Z 64.500,A 180.000,B 0.000,C 180.000} C_DIS
LIN {X 48.413,Y 94.036,Z 64.500,A 180.000,B 0.000,C 180.000} C_DIS
LIN {X 48.283,Y 94.215,Z 64.500,A 180.000,B 0.000,C 180.000} C_DIS
LIN {X 48.040,Y 94.573,Z 64.500,A 180.000,B 0.000,C 180.000} C_DIS
LIN {X 47.919,Y 94.751,Z 64.500,A 180.000,B 0.000,C 180.000} C_DIS
LIN {X 47.914,Y 94.760,Z 64.500,A 180.000,B 0.000,C 180.000} C_DIS
LIN {X 47.811,Y 94.930,Z 64.500,A 180.000,B 0.000,C 180.000} C_DIS
LIN {X 47.556,Y 95.361,Z 64.500,A 180.000,B 0.000,C 180.000} C_DIS
LIN {X 47.496,Y 95.466,Z 64.500,A 180.000,B 0.000,C 180.000} C_DIS
LIN {X 47.404,Y 95.645,Z 64.500,A 180.000,B 0.000,C 180.000} C_DIS
LIN {X 47.198,Y 96.048,Z 64.500,A 180.000,B 0.000,C 180.000} C_DIS
LIN {X 47.133,Y 96.181,Z 64.500,A 180.000,B 0.000,C 180.000} C_DIS
LIN {X 47.055,Y 96.360,Z 64.500,A 180.000,B 0.000,C 180.000} C_DIS
LIN {X 46.900,Y 96.718,Z 64.500,A 180.000,B 0.000,C 180.000} C_DIS
LIN {X 46.841,Y 96.856,Z 64.500,A 180.000,B 0.000,C 180.000} C_DIS
LIN {X 46.825,Y 96.897,Z 64.500,A 180.000,B 0.000,C 180.000} C_DIS
LIN {X 46.760,Y 97.075,Z 64.500,A 180.000,B 0.000,C 180.000} C_DIS
LIN {X 46.631,Y 97.433,Z 64.500,A 180.000,B 0.000,C 180.000} C_DIS
LIN {X 46.568,Y 97.612,Z 64.500,A 180.000,B 0.000,C 180.000} C_DIS
LIN {X 46.514,Y 97.790,Z 64.500,A 180.000,B 0.000,C 180.000} C_DIS
LIN {X 46.410,Y 98.148,Z 64.500,A 180.000,B 0.000,C 180.000} C_DIS
LIN {X 46.358,Y 98.327,Z 64.500,A 180.000,B 0.000,C 180.000} C_DIS
LIN {X 46.315,Y 98.505,Z 64.500,A 180.000,B 0.000,C 180.000} C_DIS
LIN {X 46.195,Y 99.042,Z 64.500,A 180.000,B 0.000,C 180.000} C_DIS
LIN {X 46.160,Y 99.221,Z 64.500,A 180.000,B 0.000,C 180.000} C_DIS
LIN {X 46.126,Y 99.434,Z 64.500,A 180.000,B 0.000,C 180.000} C_DIS
LIN {X 46.075,Y 99.757,Z 64.500,A 180.000,B 0.000,C 180.000} C_DIS
LIN {X 46.048,Y 99.936,Z 64.500,A 180.000,B 0.000,C 180.000} C_DIS
LIN {X 46.030,Y 100.114,Z 64.500,A 180.000,B 0.000,C 180.000} C_DIS
LIN {X 45.996,Y 100.472,Z 64.500,A 180.000,B 0.000,C 180.000} C_DIS
LIN {X 45.979,Y 100.651,Z 64.500,A 180.000,B 0.000,C 180.000} C_DIS
LIN {X 45.970,Y 100.829,Z 64.500,A 180.000,B 0.000,C 180.000} C_DIS
LIN {X 45.953,Y 101.366,Z 64.500,A 180.000,B 0.000,C 180.000} C_DIS
LIN {X 45.950,Y 101.545,Z 64.500,A 180.000,B 0.000,C 180.000} C_DIS
LIN {X 45.956,Y 101.723,Z 64.500,A 180.000,B 0.000,C 180.000} C_DIS
LIN {X 45.967,Y 102.081,Z 64.500,A 180.000,B 0.000,C 180.000} C_DIS
LIN {X 45.973,Y 102.260,Z 64.500,A 180.000,B 0.000,C 180.000} C_DIS
LIN {X 45.988,Y 102.438,Z 64.500,A 180.000,B 0.000,C 180.000} C_DIS
LIN {X 46.038,Y 102.975,Z 64.500,A 180.000,B 0.000,C 180.000} C_DIS
LIN {X 46.060,Y 103.153,Z 64.500,A 180.000,B 0.000,C 180.000} C_DIS
LIN {X 46.145,Y 103.690,Z 64.500,A 180.000,B 0.000,C 180.000} C_DIS
LIN {X 46.176,Y 103.869,Z 64.500,A 180.000,B 0.000,C 180.000} C_DIS
LIN {X 46.215,Y 104.047,Z 64.500,A 180.000,B 0.000,C 180.000} C_DIS
LIN {X 46.305,Y 104.449,Z 64.500,A 180.000,B 0.000,C 180.000} C_DIS
LIN {X 46.335,Y 104.584,Z 64.500,A 180.000,B 0.000,C 180.000} C_DIS
LIN {X 46.384,Y 104.762,Z 64.500,A 180.000,B 0.000,C 180.000} C_DIS
LIN {X 46.540,Y 105.299,Z 64.500,A 180.000,B 0.000,C 180.000} C_DIS
LIN {X 46.599,Y 105.477,Z 64.500,A 180.000,B 0.000,C 180.000} C_DIS
LIN {X 46.792,Y 106.014,Z 64.500,A 180.000,B 0.000,C 180.000} C_DIS
LIN {X 46.841,Y 106.144,Z 64.500,A 180.000,B 0.000,C 180.000} C_DIS
LIN {X 46.861,Y 106.193,Z 64.500,A 180.000,B 0.000,C 180.000} C_DIS
LIN {X 47.093,Y 106.729,Z 64.500,A 180.000,B 0.000,C 180.000} C_DIS
LIN {X 47.176,Y 106.908,Z 64.500,A 180.000,B 0.000,C 180.000} C_DIS
LIN {X 47.198,Y 106.952,Z 64.500,A 180.000,B 0.000,C 180.000} C_DIS
LIN {X 47.449,Y 107.444,Z 64.500,A 180.000,B 0.000,C 180.000} C_DIS
LIN {X 47.546,Y 107.623,Z 64.500,A 180.000,B 0.000,C 180.000} C_DIS
LIN {X 47.863,Y 108.159,Z 64.500,A 180.000,B 0.000,C 180.000} C_DIS
LIN {X 47.914,Y 108.240,Z 64.500,A 180.000,B 0.000,C 180.000} C_DIS
LIN {X 47.979,Y 108.338,Z 64.500,A 180.000,B 0.000,C 180.000} C_DIS
LIN {X 48.271,Y 108.767,Z 64.500,A 180.000,B 0.000,C 180.000} C_DIS
LIN {X 48.345,Y 108.874,Z 64.500,A 180.000,B 0.000,C 180.000} C_DIS
LIN {X 48.450,Y 109.012,Z 64.500,A 180.000,B 0.000,C 180.000} C_DIS
LIN {X 48.759,Y 109.410,Z 64.500,A 180.000,B 0.000,C 180.000} C_DIS
LIN {X 48.807,Y 109.472,Z 64.500,A 180.000,B 0.000,C 180.000} C_DIS
LIN {X 48.907,Y 109.589,Z 64.500,A 180.000,B 0.000,C 180.000} C_DIS
LIN {X 49.223,Y 109.947,Z 64.500,A 180.000,B 0.000,C 180.000} C_DIS
LIN {X 49.344,Y 110.083,Z 64.500,A 180.000,B 0.000,C 180.000} C_DIS
LIN {X 49.384,Y 110.126,Z 64.500,A 180.000,B 0.000,C 180.000} C_DIS
LIN {X 49.523,Y 110.264,Z 64.500,A 180.000,B 0.000,C 180.000} C_DIS
LIN {X 49.742,Y 110.483,Z 64.500,A 180.000,B 0.000,C 180.000} C_DIS
LIN {X 49.880,Y 110.621,Z 64.500,A 180.000,B 0.000,C 180.000} C_DIS
LIN {X 49.923,Y 110.662,Z 64.500,A 180.000,B 0.000,C 180.000} C_DIS
LIN {X 50.059,Y 110.782,Z 64.500,A 180.000,B 0.000,C 180.000} C_DIS
LIN {X 50.416,Y 111.098,Z 64.500,A 180.000,B 0.000,C 180.000} C_DIS
LIN {X 50.535,Y 111.198,Z 64.500,A 180.000,B 0.000,C 180.000} C_DIS
LIN {X 50.595,Y 111.245,Z 64.500,A 180.000,B 0.000,C 180.000} C_DIS
LIN {X 50.996,Y 111.556,Z 64.500,A 180.000,B 0.000,C 180.000} C_DIS
LIN {X 51.131,Y 111.659,Z 64.500,A 180.000,B 0.000,C 180.000} C_DIS
LIN {X 51.241,Y 111.734,Z 64.500,A 180.000,B 0.000,C 180.000} C_DIS
LIN {X 51.668,Y 112.025,Z 64.500,A 180.000,B 0.000,C 180.000} C_DIS
LIN {X 51.769,Y 112.092,Z 64.500,A 180.000,B 0.000,C 180.000} C_DIS
LIN {X 51.783,Y 112.101,Z 64.500,A 180.000,B 0.000,C 180.000} C_DIS
; Link Move Starts
LIN {X 52.053,Y 112.262,Z 64.500,A 180.000,B 0.000,C 180.000} C_DIS
LIN {X 52.324,Y 112.422,Z 64.499,A 180.000,B 0.000,C 180.000} C_DIS
LIN {X 52.601,Y 112.574,Z 64.498,A 180.000,B 0.000,C 180.000} C_DIS
LIN {X 52.881,Y 112.717,Z 64.496,A 180.000,B 0.000,C 180.000} C_DIS
LIN {X 53.163,Y 112.858,Z 64.494,A 180.000,B 0.000,C 180.000} C_DIS
LIN {X 53.451,Y 112.985,Z 64.491,A 180.000,B 0.000,C 180.000} C_DIS
LIN {X 53.740,Y 113.110,Z 64.488,A 180.000,B 0.000,C 180.000} C_DIS
LIN {X 54.033,Y 113.225,Z 64.485,A 180.000,B 0.000,C 180.000} C_DIS
LIN {X 54.330,Y 113.332,Z 64.481,A 180.000,B 0.000,C 180.000} C_DIS
LIN {X 54.627,Y 113.437,Z 64.477,A 180.000,B 0.000,C 180.000} C_DIS
LIN {X 54.929,Y 113.526,Z 64.472,A 180.000,B 0.000,C 180.000} C_DIS
LIN {X 55.080,Y 113.570,Z 64.469,A 180.000,B 0.000,C 180.000} C_DIS
LIN {X 55.231,Y 113.614,Z 64.467,A 180.000,B 0.000,C 180.000} C_DIS
LIN {X 55.383,Y 113.657,Z 64.464,A 180.000,B 0.000,C 180.000} C_DIS
LIN {X 55.536,Y 113.692,Z 64.461,A 180.000,B 0.000,C 180.000} C_DIS
LIN {X 55.690,Y 113.727,Z 64.459,A 180.000,B 0.000,C 180.000} C_DIS
LIN {X 55.844,Y 113.761,Z 64.456,A 180.000,B 0.000,C 180.000} C_DIS
LIN {X 55.998,Y 113.795,Z 64.452,A 180.000,B 0.000,C 180.000} C_DIS
LIN {X 56.152,Y 113.828,Z 64.449,A 180.000,B 0.000,C 180.000} C_DIS
LIN {X 56.307,Y 113.854,Z 64.446,A 180.000,B 0.000,C 180.000} C_DIS
LIN {X 56.462,Y 113.879,Z 64.443,A 180.000,B 0.000,C 180.000} C_DIS
LIN {X 56.618,Y 113.903,Z 64.439,A 180.000,B 0.000,C 180.000} C_DIS
LIN {X 56.774,Y 113.928,Z 64.436,A 180.000,B 0.000,C 180.000} C_DIS
LIN {X 56.929,Y 113.951,Z 64.432,A 180.000,B 0.000,C 180.000} C_DIS
LIN {X 57.086,Y 113.967,Z 64.428,A 180.000,B 0.000,C 180.000} C_DIS
LIN {X 57.243,Y 113.982,Z 64.425,A 180.000,B 0.000,C 180.000} C_DIS
LIN {X 57.400,Y 113.997,Z 64.421,A 180.000,B 0.000,C 180.000} C_DIS
LIN {X 57.556,Y 114.012,Z 64.417,A 180.000,B 0.000,C 180.000} C_DIS
LIN {X 57.713,Y 114.025,Z 64.413,A 180.000,B 0.000,C 180.000} C_DIS
LIN {X 57.871,Y 114.031,Z 64.409,A 180.000,B 0.000,C 180.000} C_DIS
LIN {X 58.028,Y 114.036,Z 64.405,A 180.000,B 0.000,C 180.000} C_DIS
LIN {X 58.186,Y 114.041,Z 64.400,A 180.000,B 0.000,C 180.000} C_DIS
LIN {X 58.343,Y 114.046,Z 64.396,A 180.000,B 0.000,C 180.000} C_DIS
LIN {X 58.500,Y 114.050,Z 64.392,A 180.000,B 0.000,C 180.000} C_DIS
LIN {X 58.658,Y 114.046,Z 64.387,A 180.000,B 0.000,C 180.000} C_DIS
LIN {X 58.815,Y 114.041,Z 64.383,A 180.000,B 0.000,C 180.000} C_DIS
LIN {X 58.973,Y 114.036,Z 64.378,A 180.000,B 0.000,C 180.000} C_DIS
LIN {X 59.130,Y 114.031,Z 64.373,A 180.000,B 0.000,C 180.000} C_DIS
LIN {X 59.288,Y 114.025,Z 64.369,A 180.000,B 0.000,C 180.000} C_DIS
LIN {X 59.445,Y 114.012,Z 64.364,A 180.000,B 0.000,C 180.000} C_DIS
LIN {X 59.601,Y 113.997,Z 64.359,A 180.000,B 0.000,C 180.000} C_DIS
LIN {X 59.758,Y 113.982,Z 64.354,A 180.000,B 0.000,C 180.000} C_DIS
LIN {X 59.837,Y 113.975,Z 64.351,A 180.000,B 0.000,C 180.000} C_DIS
LIN {X 59.915,Y 113.967,Z 64.349,A 180.000,B 0.000,C 180.000} C_DIS
LIN {X 59.993,Y 113.960,Z 64.346,A 180.000,B 0.000,C 180.000} C_DIS
LIN {X 60.072,Y 113.951,Z 64.344,A 180.000,B 0.000,C 180.000} C_DIS
LIN {X 60.150,Y 113.940,Z 64.341,A 180.000,B 0.000,C 180.000} C_DIS
LIN {X 60.227,Y 113.928,Z 64.339,A 180.000,B 0.000,C 180.000} C_DIS
LIN {X 60.305,Y 113.916,Z 64.336,A 180.000,B 0.000,C 180.000} C_DIS
LIN {X 60.461,Y 113.891,Z 64.331,A 180.000,B 0.000,C 180.000} C_DIS
LIN {X 60.616,Y 113.866,Z 64.325,A 180.000,B 0.000,C 180.000} C_DIS
LIN {X 60.772,Y 113.842,Z 64.320,A 180.000,B 0.000,C 180.000} C_DIS
LIN {X 60.849,Y 113.828,Z 64.317,A 180.000,B 0.000,C 180.000} C_DIS
LIN {X 60.927,Y 113.812,Z 64.315,A 180.000,B 0.000,C 180.000} C_DIS
LIN {X 61.080,Y 113.778,Z 64.309,A 180.000,B 0.000,C 180.000} C_DIS
LIN {X 61.157,Y 113.761,Z 64.307,A 180.000,B 0.000,C 180.000} C_DIS
LIN {X 61.311,Y 113.726,Z 64.301,A 180.000,B 0.000,C 180.000} C_DIS
LIN {X 61.541,Y 113.675,Z 64.293,A 180.000,B 0.000,C 180.000} C_DIS
LIN {X 61.618,Y 113.657,Z 64.290,A 180.000,B 0.000,C 180.000} C_DIS
LIN {X 61.694,Y 113.636,Z 64.287,A 180.000,B 0.000,C 180.000} C_DIS
LIN {X 61.770,Y 113.614,Z 64.285,A 180.000,B 0.000,C 180.000} C_DIS
LIN {X 61.921,Y 113.570,Z 64.279,A 180.000,B 0.000,C 180.000} C_DIS
LIN {X 62.148,Y 113.504,Z 64.271,A 180.000,B 0.000,C 180.000} C_DIS
LIN {X 62.299,Y 113.460,Z 64.265,A 180.000,B 0.000,C 180.000} C_DIS
LIN {X 62.374,Y 113.437,Z 64.263,A 180.000,B 0.000,C 180.000} C_DIS
LIN {X 62.449,Y 113.412,Z 64.260,A 180.000,B 0.000,C 180.000} C_DIS
LIN {X 62.597,Y 113.358,Z 64.254,A 180.000,B 0.000,C 180.000} C_DIS
LIN {X 62.671,Y 113.332,Z 64.252,A 180.000,B 0.000,C 180.000} C_DIS
LIN {X 62.819,Y 113.278,Z 64.246,A 180.000,B 0.000,C 180.000} C_DIS
LIN {X 63.042,Y 113.198,Z 64.238,A 180.000,B 0.000,C 180.000} C_DIS
LIN {X 63.115,Y 113.171,Z 64.235,A 180.000,B 0.000,C 180.000} C_DIS
LIN {X 63.188,Y 113.141,Z 64.232,A 180.000,B 0.000,C 180.000} C_DIS
LIN {X 63.260,Y 113.109,Z 64.230,A 180.000,B 0.000,C 180.000} C_DIS
LIN {X 63.405,Y 113.047,Z 64.224,A 180.000,B 0.000,C 180.000} C_DIS
LIN {X 63.766,Y 112.890,Z 64.210,A 180.000,B 0.000,C 180.000} C_DIS
LIN {X 63.838,Y 112.858,Z 64.208,A 180.000,B 0.000,C 180.000} C_DIS
LIN {X 63.909,Y 112.824,Z 64.205,A 180.000,B 0.000,C 180.000} C_DIS
LIN {X 64.049,Y 112.752,Z 64.199,A 180.000,B 0.000,C 180.000} C_DIS
LIN {X 64.119,Y 112.716,Z 64.197,A 180.000,B 0.000,C 180.000} C_DIS
LIN {X 64.260,Y 112.645,Z 64.191,A 180.000,B 0.000,C 180.000} C_DIS
LIN {X 64.470,Y 112.538,Z 64.183,A 180.000,B 0.000,C 180.000} C_DIS
LIN {X 64.540,Y 112.501,Z 64.180,A 180.000,B 0.000,C 180.000} C_DIS
LIN {X 64.609,Y 112.462,Z 64.177,A 180.000,B 0.000,C 180.000} C_DIS
LIN {X 64.676,Y 112.422,Z 64.175,A 180.000,B 0.000,C 180.000} C_DIS
LIN {X 64.812,Y 112.342,Z 64.169,A 180.000,B 0.000,C 180.000} C_DIS
LIN {X 65.151,Y 112.141,Z 64.155,A 180.000,B 0.000,C 180.000} C_DIS
LIN {X 65.218,Y 112.100,Z 64.153,A 180.000,B 0.000,C 180.000} C_DIS
LIN {X 65.284,Y 112.057,Z 64.150,A 180.000,B 0.000,C 180.000} C_DIS
LIN {X 65.414,Y 111.969,Z 64.144,A 180.000,B 0.000,C 180.000} C_DIS
LIN {X 65.545,Y 111.880,Z 64.139,A 180.000,B 0.000,C 180.000} C_DIS
LIN {X 65.805,Y 111.703,Z 64.128,A 180.000,B 0.000,C 180.000} C_DIS
LIN {X 65.870,Y 111.658,Z 64.125,A 180.000,B 0.000,C 180.000} C_DIS
LIN {X 65.933,Y 111.611,Z 64.122,A 180.000,B 0.000,C 180.000} C_DIS
LIN {X 65.995,Y 111.563,Z 64.120,A 180.000,B 0.000,C 180.000} C_DIS
LIN {X 66.182,Y 111.418,Z 64.111,A 180.000,B 0.000,C 180.000} C_DIS
LIN {X 66.306,Y 111.322,Z 64.106,A 180.000,B 0.000,C 180.000} C_DIS
LIN {X 66.431,Y 111.225,Z 64.100,A 180.000,B 0.000,C 180.000} C_DIS
LIN {X 66.492,Y 111.176,Z 64.098,A 180.000,B 0.000,C 180.000} C_DIS
LIN {X 66.552,Y 111.125,Z 64.095,A 180.000,B 0.000,C 180.000} C_DIS
LIN {X 66.611,Y 111.073,Z 64.092,A 180.000,B 0.000,C 180.000} C_DIS
LIN {X 67.025,Y 110.709,Z 64.073,A 180.000,B 0.000,C 180.000} C_DIS
LIN {X 67.083,Y 110.656,Z 64.070,A 180.000,B 0.000,C 180.000} C_DIS
LIN {X 67.140,Y 110.601,Z 64.067,A 180.000,B 0.000,C 180.000} C_DIS
LIN {X 67.196,Y 110.546,Z 64.065,A 180.000,B 0.000,C 180.000} C_DIS
LIN {X 67.530,Y 110.211,Z 64.048,A 180.000,B 0.000,C 180.000} C_DIS
LIN {X 67.586,Y 110.156,Z 64.045,A 180.000,B 0.000,C 180.000} C_DIS
LIN {X 67.641,Y 110.099,Z 64.043,A 180.000,B 0.000,C 180.000} C_DIS
LIN {X 67.694,Y 110.041,Z 64.040,A 180.000,B 0.000,C 180.000} C_DIS
LIN {X 67.746,Y 109.982,Z 64.037,A 180.000,B 0.000,C 180.000} C_DIS
LIN {X 68.111,Y 109.569,Z 64.018,A 180.000,B 0.000,C 180.000} C_DIS
LIN {X 68.162,Y 109.509,Z 64.015,A 180.000,B 0.000,C 180.000} C_DIS
LIN {X 68.212,Y 109.448,Z 64.012,A 180.000,B 0.000,C 180.000} C_DIS
LIN {X 68.260,Y 109.386,Z 64.010,A 180.000,B 0.000,C 180.000} C_DIS
LIN {X 68.598,Y 108.950,Z 63.990,A 180.000,B 0.000,C 180.000} C_DIS
LIN {X 68.645,Y 108.887,Z 63.988,A 180.000,B 0.000,C 180.000} C_DIS
LIN {X 68.691,Y 108.823,Z 63.985,A 180.000,B 0.000,C 180.000} C_DIS
LIN {X 68.735,Y 108.758,Z 63.982,A 180.000,B 0.000,C 180.000} C_DIS
LIN {X 69.045,Y 108.302,Z 63.963,A 180.000,B 0.000,C 180.000} C_DIS
LIN {X 69.089,Y 108.237,Z 63.960,A 180.000,B 0.000,C 180.000} C_DIS
LIN {X 69.130,Y 108.170,Z 63.957,A 180.000,B 0.000,C 180.000} C_DIS
LIN {X 69.170,Y 108.102,Z 63.955,A 180.000,B 0.000,C 180.000} C_DIS
LIN {X 69.451,Y 107.627,Z 63.935,A 180.000,B 0.000,C 180.000} C_DIS
LIN {X 69.490,Y 107.559,Z 63.933,A 180.000,B 0.000,C 180.000} C_DIS
LIN {X 69.528,Y 107.490,Z 63.930,A 180.000,B 0.000,C 180.000} C_DIS
LIN {X 69.563,Y 107.420,Z 63.927,A 180.000,B 0.000,C 180.000} C_DIS
LIN {X 69.814,Y 106.928,Z 63.908,A 180.000,B 0.000,C 180.000} C_DIS
LIN {X 69.849,Y 106.858,Z 63.905,A 180.000,B 0.000,C 180.000} C_DIS
LIN {X 69.882,Y 106.786,Z 63.902,A 180.000,B 0.000,C 180.000} C_DIS
LIN {X 69.913,Y 106.714,Z 63.900,A 180.000,B 0.000,C 180.000} C_DIS
LIN {X 70.007,Y 106.497,Z 63.891,A 180.000,B 0.000,C 180.000} C_DIS
LIN {X 70.069,Y 106.353,Z 63.886,A 180.000,B 0.000,C 180.000} C_DIS
LIN {X 70.132,Y 106.208,Z 63.880,A 180.000,B 0.000,C 180.000} C_DIS
LIN {X 70.162,Y 106.136,Z 63.878,A 180.000,B 0.000,C 180.000} C_DIS
LIN {X 70.191,Y 106.062,Z 63.875,A 180.000,B 0.000,C 180.000} C_DIS
LIN {X 70.217,Y 105.988,Z 63.872,A 180.000,B 0.000,C 180.000} C_DIS
LIN {X 70.404,Y 105.469,Z 63.853,A 180.000,B 0.000,C 180.000} C_DIS
LIN {X 70.430,Y 105.395,Z 63.850,A 180.000,B 0.000,C 180.000} C_DIS
LIN {X 70.454,Y 105.320,Z 63.847,A 180.000,B 0.000,C 180.000} C_DIS
LIN {X 70.476,Y 105.244,Z 63.845,A 180.000,B 0.000,C 180.000} C_DIS
LIN {X 70.542,Y 105.017,Z 63.836,A 180.000,B 0.000,C 180.000} C_DIS
LIN {X 70.564,Y 104.942,Z 63.834,A 180.000,B 0.000,C 180.000} C_DIS
LIN {X 70.608,Y 104.791,Z 63.828,A 180.000,B 0.000,C 180.000} C_DIS
LIN {X 70.630,Y 104.715,Z 63.825,A 180.000,B 0.000,C 180.000} C_DIS
LIN {X 70.651,Y 104.639,Z 63.823,A 180.000,B 0.000,C 180.000} C_DIS
LIN {X 70.670,Y 104.563,Z 63.820,A 180.000,B 0.000,C 180.000} C_DIS
LIN {X 70.687,Y 104.486,Z 63.817,A 180.000,B 0.000,C 180.000} C_DIS
LIN {X 70.790,Y 104.025,Z 63.801,A 180.000,B 0.000,C 180.000} C_DIS
LIN {X 70.807,Y 103.948,Z 63.798,A 180.000,B 0.000,C 180.000} C_DIS
LIN {X 70.824,Y 103.871,Z 63.795,A 180.000,B 0.000,C 180.000} C_DIS
LIN {X 70.838,Y 103.793,Z 63.792,A 180.000,B 0.000,C 180.000} C_DIS
LIN {X 70.850,Y 103.716,Z 63.790,A 180.000,B 0.000,C 180.000} C_DIS
LIN {X 70.875,Y 103.560,Z 63.784,A 180.000,B 0.000,C 180.000} C_DIS
LIN {X 70.912,Y 103.327,Z 63.776,A 180.000,B 0.000,C 180.000} C_DIS
LIN {X 70.937,Y 103.171,Z 63.770,A 180.000,B 0.000,C 180.000} C_DIS
LIN {X 70.948,Y 103.093,Z 63.768,A 180.000,B 0.000,C 180.000} C_DIS
LIN {X 70.958,Y 103.015,Z 63.765,A 180.000,B 0.000,C 180.000} C_DIS
LIN {X 70.965,Y 102.937,Z 63.762,A 180.000,B 0.000,C 180.000} C_DIS
LIN {X 70.987,Y 102.701,Z 63.754,A 180.000,B 0.000,C 180.000} C_DIS
LIN {X 71.002,Y 102.545,Z 63.748,A 180.000,B 0.000,C 180.000} C_DIS
LIN {X 71.010,Y 102.466,Z 63.746,A 180.000,B 0.000,C 180.000} C_DIS
LIN {X 71.017,Y 102.388,Z 63.743,A 180.000,B 0.000,C 180.000} C_DIS
LIN {X 71.024,Y 102.309,Z 63.740,A 180.000,B 0.000,C 180.000} C_DIS
LIN {X 71.028,Y 102.231,Z 63.737,A 180.000,B 0.000,C 180.000} C_DIS
LIN {X 71.031,Y 102.152,Z 63.735,A 180.000,B 0.000,C 180.000} C_DIS
LIN {X 71.036,Y 101.995,Z 63.729,A 180.000,B 0.000,C 180.000} C_DIS
LIN {X 71.043,Y 101.758,Z 63.721,A 180.000,B 0.000,C 180.000} C_DIS
LIN {X 71.048,Y 101.601,Z 63.715,A 180.000,B 0.000,C 180.000} C_DIS
LIN {X 71.050,Y 101.522,Z 63.713,A 180.000,B 0.000,C 180.000} C_DIS
LIN {X 71.049,Y 101.444,Z 63.710,A 180.000,B 0.000,C 180.000} C_DIS
LIN {X 71.047,Y 101.365,Z 63.707,A 180.000,B 0.000,C 180.000} C_DIS
LIN {X 71.040,Y 101.129,Z 63.699,A 180.000,B 0.000,C 180.000} C_DIS
LIN {X 71.035,Y 100.971,Z 63.693,A 180.000,B 0.000,C 180.000} C_DIS
LIN {X 71.030,Y 100.814,Z 63.688,A 180.000,B 0.000,C 180.000} C_DIS
LIN {X 71.027,Y 100.735,Z 63.685,A 180.000,B 0.000,C 180.000} C_DIS
LIN {X 71.021,Y 100.657,Z 63.682,A 180.000,B 0.000,C 180.000} C_DIS
LIN {X 71.014,Y 100.578,Z 63.680,A 180.000,B 0.000,C 180.000} C_DIS
LIN {X 70.999,Y 100.421,Z 63.674,A 180.000,B 0.000,C 180.000} C_DIS
LIN {X 70.984,Y 100.265,Z 63.669,A 180.000,B 0.000,C 180.000} C_DIS
LIN {X 70.969,Y 100.108,Z 63.664,A 180.000,B 0.000,C 180.000} C_DIS
LIN {X 70.962,Y 100.029,Z 63.661,A 180.000,B 0.000,C 180.000} C_DIS
LIN {X 70.954,Y 99.951,Z 63.659,A 180.000,B 0.000,C 180.000} C_DIS
LIN {X 70.944,Y 99.873,Z 63.656,A 180.000,B 0.000,C 180.000} C_DIS
LIN {X 70.931,Y 99.795,Z 63.654,A 180.000,B 0.000,C 180.000} C_DIS
LIN {X 70.919,Y 99.717,Z 63.651,A 180.000,B 0.000,C 180.000} C_DIS
LIN {X 70.907,Y 99.640,Z 63.649,A 180.000,B 0.000,C 180.000} C_DIS
LIN {X 70.882,Y 99.484,Z 63.644,A 180.000,B 0.000,C 180.000} C_DIS
LIN {X 70.857,Y 99.329,Z 63.639,A 180.000,B 0.000,C 180.000} C_DIS
LIN {X 70.832,Y 99.173,Z 63.634,A 180.000,B 0.000,C 180.000} C_DIS
LIN {X 70.800,Y 99.019,Z 63.629,A 180.000,B 0.000,C 180.000} C_DIS
LIN {X 70.766,Y 98.865,Z 63.624,A 180.000,B 0.000,C 180.000} C_DIS
LIN {X 70.731,Y 98.711,Z 63.620,A 180.000,B 0.000,C 180.000} C_DIS
LIN {X 70.697,Y 98.558,Z 63.615,A 180.000,B 0.000,C 180.000} C_DIS
LIN {X 70.662,Y 98.404,Z 63.611,A 180.000,B 0.000,C 180.000} C_DIS
LIN {X 70.620,Y 98.252,Z 63.606,A 180.000,B 0.000,C 180.000} C_DIS
LIN {X 70.576,Y 98.101,Z 63.602,A 180.000,B 0.000,C 180.000} C_DIS
LIN {X 70.532,Y 97.950,Z 63.597,A 180.000,B 0.000,C 180.000} C_DIS
LIN {X 70.488,Y 97.799,Z 63.593,A 180.000,B 0.000,C 180.000} C_DIS
LIN {X 70.444,Y 97.647,Z 63.589,A 180.000,B 0.000,C 180.000} C_DIS
LIN {X 70.393,Y 97.499,Z 63.585,A 180.000,B 0.000,C 180.000} C_DIS
LIN {X 70.339,Y 97.350,Z 63.581,A 180.000,B 0.000,C 180.000} C_DIS
LIN {X 70.286,Y 97.202,Z 63.577,A 180.000,B 0.000,C 180.000} C_DIS
LIN {X 70.233,Y 97.054,Z 63.573,A 180.000,B 0.000,C 180.000} C_DIS
LIN {X 70.179,Y 96.906,Z 63.570,A 180.000,B 0.000,C 180.000} C_DIS
LIN {X 70.118,Y 96.761,Z 63.566,A 180.000,B 0.000,C 180.000} C_DIS
LIN {X 70.056,Y 96.616,Z 63.562,A 180.000,B 0.000,C 180.000} C_DIS
LIN {X 69.993,Y 96.471,Z 63.559,A 180.000,B 0.000,C 180.000} C_DIS
LIN {X 69.931,Y 96.327,Z 63.556,A 180.000,B 0.000,C 180.000} C_DIS
LIN {X 69.868,Y 96.183,Z 63.552,A 180.000,B 0.000,C 180.000} C_DIS
LIN {X 69.798,Y 96.041,Z 63.549,A 180.000,B 0.000,C 180.000} C_DIS
LIN {X 69.727,Y 95.901,Z 63.546,A 180.000,B 0.000,C 180.000} C_DIS
LIN {X 69.655,Y 95.761,Z 63.543,A 180.000,B 0.000,C 180.000} C_DIS
LIN {X 69.584,Y 95.620,Z 63.540,A 180.000,B 0.000,C 180.000} C_DIS
LIN {X 69.512,Y 95.480,Z 63.537,A 180.000,B 0.000,C 180.000} C_DIS
LIN {X 69.434,Y 95.343,Z 63.534,A 180.000,B 0.000,C 180.000} C_DIS
LIN {X 69.353,Y 95.208,Z 63.532,A 180.000,B 0.000,C 180.000} C_DIS
LIN {X 69.273,Y 95.072,Z 63.529,A 180.000,B 0.000,C 180.000} C_DIS
LIN {X 69.193,Y 94.937,Z 63.527,A 180.000,B 0.000,C 180.000} C_DIS
LIN {X 69.026,Y 94.670,Z 63.522,A 180.000,B 0.000,C 180.000} C_DIS
LIN {X 68.849,Y 94.409,Z 63.518,A 180.000,B 0.000,C 180.000} C_DIS
LIN {X 68.672,Y 94.149,Z 63.514,A 180.000,B 0.000,C 180.000} C_DIS
LIN {X 68.480,Y 93.899,Z 63.511,A 180.000,B 0.000,C 180.000} C_DIS
LIN {X 68.287,Y 93.650,Z 63.508,A 180.000,B 0.000,C 180.000} C_DIS
LIN {X 68.088,Y 93.406,Z 63.505,A 180.000,B 0.000,C 180.000} C_DIS
LIN {X 67.880,Y 93.169,Z 63.503,A 180.000,B 0.000,C 180.000} C_DIS
LIN {X 67.671,Y 92.933,Z 63.502,A 180.000,B 0.000,C 180.000} C_DIS
LIN {X 67.450,Y 92.709,Z 63.501,A 180.000,B 0.000,C 180.000} C_DIS
LIN {X 67.228,Y 92.486,Z 63.500,A 180.000,B 0.000,C 180.000} C_DIS
LIN {X 67.061,Y 92.325,Z 63.500,A 180.000,B 0.000,C 180.000} C_DIS
; Cutting Move Starts
LIN {X 67.042,Y 92.307,Z 63.500,A 180.000,B 0.000,C 180.000} C_DIS
LIN {X 66.976,Y 92.249,Z 63.500,A 180.000,B 0.000,C 180.000} C_DIS
LIN {X 66.571,Y 91.891,Z 63.500,A 180.000,B 0.000,C 180.000} C_DIS
LIN {X 66.506,Y 91.835,Z 63.500,A 180.000,B 0.000,C 180.000} C_DIS
LIN {X 66.350,Y 91.712,Z 63.500,A 180.000,B 0.000,C 180.000} C_DIS
LIN {X 65.969,Y 91.417,Z 63.500,A 180.000,B 0.000,C 180.000} C_DIS
LIN {X 65.887,Y 91.355,Z 63.500,A 180.000,B 0.000,C 180.000} C_DIS
LIN {X 65.791,Y 91.287,Z 63.500,A 180.000,B 0.000,C 180.000} C_DIS
LIN {X 65.364,Y 90.997,Z 63.500,A 180.000,B 0.000,C 180.000} C_DIS
LIN {X 65.254,Y 90.923,Z 63.500,A 180.000,B 0.000,C 180.000} C_DIS
LIN {X 65.083,Y 90.818,Z 63.500,A 180.000,B 0.000,C 180.000} C_DIS
LIN {X 64.718,Y 90.603,Z 63.500,A 180.000,B 0.000,C 180.000} C_DIS
LIN {X 64.539,Y 90.499,Z 63.500,A 180.000,B 0.000,C 180.000} C_DIS
LIN {X 64.467,Y 90.461,Z 63.500,A 180.000,B 0.000,C 180.000} C_DIS
LIN {X 64.003,Y 90.224,Z 63.500,A 180.000,B 0.000,C 180.000} C_DIS
LIN {X 63.824,Y 90.135,Z 63.500,A 180.000,B 0.000,C 180.000} C_DIS
LIN {X 63.752,Y 90.103,Z 63.500,A 180.000,B 0.000,C 180.000} C_DIS
LIN {X 63.288,Y 89.903,Z 63.500,A 180.000,B 0.000,C 180.000} C_DIS
LIN {X 63.109,Y 89.827,Z 63.500,A 180.000,B 0.000,C 180.000} C_DIS
LIN {X 62.930,Y 89.762,Z 63.500,A 180.000,B 0.000,C 180.000} C_DIS
LIN {X 62.573,Y 89.633,Z 63.500,A 180.000,B 0.000,C 180.000} C_DIS
LIN {X 62.394,Y 89.569,Z 63.500,A 180.000,B 0.000,C 180.000} C_DIS
LIN {X 62.387,Y 89.567,Z 63.500,A 180.000,B 0.000,C 180.000} C_DIS
LIN {X 62.215,Y 89.516,Z 63.500,A 180.000,B 0.000,C 180.000} C_DIS
LIN {X 61.777,Y 89.388,Z 63.500,A 180.000,B 0.000,C 180.000} C_DIS
LIN {X 61.679,Y 89.360,Z 63.500,A 180.000,B 0.000,C 180.000} C_DIS
LIN {X 61.500,Y 89.316,Z 63.500,A 180.000,B 0.000,C 180.000} C_DIS
LIN {X 60.964,Y 89.196,Z 63.500,A 180.000,B 0.000,C 180.000} C_DIS
LIN {X 60.785,Y 89.161,Z 63.500,A 180.000,B 0.000,C 180.000} C_DIS
LIN {X 60.606,Y 89.132,Z 63.500,A 180.000,B 0.000,C 180.000} C_DIS
LIN {X 60.249,Y 89.076,Z 63.500,A 180.000,B 0.000,C 180.000} C_DIS
LIN {X 60.070,Y 89.049,Z 63.500,A 180.000,B 0.000,C 180.000} C_DIS
LIN {X 59.892,Y 89.031,Z 63.500,A 180.000,B 0.000,C 180.000} C_DIS
LIN {X 59.534,Y 88.997,Z 63.500,A 180.000,B 0.000,C 180.000} C_DIS
LIN {X 59.355,Y 88.980,Z 63.500,A 180.000,B 0.000,C 180.000} C_DIS
LIN {X 59.176,Y 88.970,Z 63.500,A 180.000,B 0.000,C 180.000} C_DIS
LIN {X 58.640,Y 88.953,Z 63.500,A 180.000,B 0.000,C 180.000} C_DIS
LIN {X 58.461,Y 88.950,Z 63.500,A 180.000,B 0.000,C 180.000} C_DIS
LIN {X 58.282,Y 88.956,Z 63.500,A 180.000,B 0.000,C 180.000} C_DIS
LIN {X 57.925,Y 88.967,Z 63.500,A 180.000,B 0.000,C 180.000} C_DIS
LIN {X 57.746,Y 88.973,Z 63.500,A 180.000,B 0.000,C 180.000} C_DIS
LIN {X 57.567,Y 88.987,Z 63.500,A 180.000,B 0.000,C 180.000} C_DIS
LIN {X 57.031,Y 89.038,Z 63.500,A 180.000,B 0.000,C 180.000} C_DIS
LIN {X 56.852,Y 89.060,Z 63.500,A 180.000,B 0.000,C 180.000} C_DIS
LIN {X 56.316,Y 89.145,Z 63.500,A 180.000,B 0.000,C 180.000} C_DIS
LIN {X 56.137,Y 89.174,Z 63.500,A 180.000,B 0.000,C 180.000} C_DIS
LIN {X 55.977,Y 89.209,Z 63.500,A 180.000,B 0.000,C 180.000} C_DIS
LIN {X 55.601,Y 89.293,Z 63.500,A 180.000,B 0.000,C 180.000} C_DIS
LIN {X 55.422,Y 89.334,Z 63.500,A 180.000,B 0.000,C 180.000} C_DIS
LIN {X 55.243,Y 89.382,Z 63.500,A 180.000,B 0.000,C 180.000} C_DIS
LIN {X 54.707,Y 89.538,Z 63.500,A 180.000,B 0.000,C 180.000} C_DIS
LIN {X 54.613,Y 89.567,Z 63.500,A 180.000,B 0.000,C 180.000} C_DIS
LIN {X 54.528,Y 89.597,Z 63.500,A 180.000,B 0.000,C 180.000} C_DIS
LIN {X 53.992,Y 89.790,Z 63.500,A 180.000,B 0.000,C 180.000} C_DIS
LIN {X 53.813,Y 89.859,Z 63.500,A 180.000,B 0.000,C 180.000} C_DIS
LIN {X 53.455,Y 90.014,Z 63.500,A 180.000,B 0.000,C 180.000} C_DIS
LIN {X 53.248,Y 90.103,Z 63.500,A 180.000,B 0.000,C 180.000} C_DIS
LIN {X 53.098,Y 90.173,Z 63.500,A 180.000,B 0.000,C 180.000} C_DIS
LIN {X 52.919,Y 90.264,Z 63.500,A 180.000,B 0.000,C 180.000} C_DIS
LIN {X 52.533,Y 90.461,Z 63.500,A 180.000,B 0.000,C 180.000} C_DIS
LIN {X 52.383,Y 90.543,Z 63.500,A 180.000,B 0.000,C 180.000} C_DIS
LIN {X 51.847,Y 90.860,Z 63.500,A 180.000,B 0.000,C 180.000} C_DIS
LIN {X 51.668,Y 90.975,Z 63.500,A 180.000,B 0.000,C 180.000} C_DIS
LIN {X 51.310,Y 91.218,Z 63.500,A 180.000,B 0.000,C 180.000} C_DIS
LIN {X 51.131,Y 91.341,Z 63.500,A 180.000,B 0.000,C 180.000} C_DIS
LIN {X 51.113,Y 91.355,Z 63.500,A 180.000,B 0.000,C 180.000} C_DIS
LIN {X 50.953,Y 91.478,Z 63.500,A 180.000,B 0.000,C 180.000} C_DIS
LIN {X 50.595,Y 91.755,Z 63.500,A 180.000,B 0.000,C 180.000} C_DIS
LIN {X 50.429,Y 91.891,Z 63.500,A 180.000,B 0.000,C 180.000} C_DIS
LIN {X 50.024,Y 92.249,Z 63.500,A 180.000,B 0.000,C 180.000} C_DIS
LIN {X 49.880,Y 92.379,Z 63.500,A 180.000,B 0.000,C 180.000} C_DIS
LIN {X 49.831,Y 92.427,Z 63.500,A 180.000,B 0.000,C 180.000} C_DIS
LIN {X 49.474,Y 92.785,Z 63.500,A 180.000,B 0.000,C 180.000} C_DIS
LIN {X 49.344,Y 92.917,Z 63.500,A 180.000,B 0.000,C 180.000} C_DIS
LIN {X 49.302,Y 92.964,Z 63.500,A 180.000,B 0.000,C 180.000} C_DIS
LIN {X 48.986,Y 93.321,Z 63.500,A 180.000,B 0.000,C 180.000} C_DIS
LIN {X 48.830,Y 93.500,Z 63.500,A 180.000,B 0.000,C 180.000} C_DIS
LIN {X 48.807,Y 93.528,Z 63.500,A 180.000,B 0.000,C 180.000} C_DIS
LIN {X 48.690,Y 93.679,Z 63.500,A 180.000,B 0.000,C 180.000} C_DIS
LIN {X 48.413,Y 94.036,Z 63.500,A 180.000,B 0.000,C 180.000} C_DIS
LIN {X 48.283,Y 94.215,Z 63.500,A 180.000,B 0.000,C 180.000} C_DIS
LIN {X 48.040,Y 94.573,Z 63.500,A 180.000,B 0.000,C 180.000} C_DIS
LIN {X 47.919,Y 94.751,Z 63.500,A 180.000,B 0.000,C 180.000} C_DIS
LIN {X 47.914,Y 94.760,Z 63.500,A 180.000,B 0.000,C 180.000} C_DIS
LIN {X 47.811,Y 94.930,Z 63.500,A 180.000,B 0.000,C 180.000} C_DIS
LIN {X 47.556,Y 95.361,Z 63.500,A 180.000,B 0.000,C 180.000} C_DIS
LIN {X 47.496,Y 95.466,Z 63.500,A 180.000,B 0.000,C 180.000} C_DIS
LIN {X 47.404,Y 95.645,Z 63.500,A 180.000,B 0.000,C 180.000} C_DIS
LIN {X 47.198,Y 96.048,Z 63.500,A 180.000,B 0.000,C 180.000} C_DIS
LIN {X 47.133,Y 96.181,Z 63.500,A 180.000,B 0.000,C 180.000} C_DIS
LIN {X 47.055,Y 96.360,Z 63.500,A 180.000,B 0.000,C 180.000} C_DIS
LIN {X 46.900,Y 96.718,Z 63.500,A 180.000,B 0.000,C 180.000} C_DIS
LIN {X 46.841,Y 96.856,Z 63.500,A 180.000,B 0.000,C 180.000} C_DIS
LIN {X 46.825,Y 96.897,Z 63.500,A 180.000,B 0.000,C 180.000} C_DIS
LIN {X 46.760,Y 97.075,Z 63.500,A 180.000,B 0.000,C 180.000} C_DIS
LIN {X 46.631,Y 97.433,Z 63.500,A 180.000,B 0.000,C 180.000} C_DIS
LIN {X 46.568,Y 97.612,Z 63.500,A 180.000,B 0.000,C 180.000} C_DIS
LIN {X 46.514,Y 97.790,Z 63.500,A 180.000,B 0.000,C 180.000} C_DIS
LIN {X 46.410,Y 98.148,Z 63.500,A 180.000,B 0.000,C 180.000} C_DIS
LIN {X 46.358,Y 98.327,Z 63.500,A 180.000,B 0.000,C 180.000} C_DIS
LIN {X 46.315,Y 98.505,Z 63.500,A 180.000,B 0.000,C 180.000} C_DIS
LIN {X 46.195,Y 99.042,Z 63.500,A 180.000,B 0.000,C 180.000} C_DIS
LIN {X 46.160,Y 99.221,Z 63.500,A 180.000,B 0.000,C 180.000} C_DIS
LIN {X 46.126,Y 99.434,Z 63.500,A 180.000,B 0.000,C 180.000} C_DIS
LIN {X 46.075,Y 99.757,Z 63.500,A 180.000,B 0.000,C 180.000} C_DIS
LIN {X 46.048,Y 99.936,Z 63.500,A 180.000,B 0.000,C 180.000} C_DIS
LIN {X 46.030,Y 100.114,Z 63.500,A 180.000,B 0.000,C 180.000} C_DIS
LIN {X 45.996,Y 100.472,Z 63.500,A 180.000,B 0.000,C 180.000} C_DIS
LIN {X 45.979,Y 100.651,Z 63.500,A 180.000,B 0.000,C 180.000} C_DIS
LIN {X 45.970,Y 100.829,Z 63.500,A 180.000,B 0.000,C 180.000} C_DIS
LIN {X 45.953,Y 101.366,Z 63.500,A 180.000,B 0.000,C 180.000} C_DIS
LIN {X 45.950,Y 101.545,Z 63.500,A 180.000,B 0.000,C 180.000} C_DIS
LIN {X 45.956,Y 101.723,Z 63.500,A 180.000,B 0.000,C 180.000} C_DIS
LIN {X 45.967,Y 102.081,Z 63.500,A 180.000,B 0.000,C 180.000} C_DIS
LIN {X 45.973,Y 102.260,Z 63.500,A 180.000,B 0.000,C 180.000} C_DIS
LIN {X 45.988,Y 102.438,Z 63.500,A 180.000,B 0.000,C 180.000} C_DIS
LIN {X 46.038,Y 102.975,Z 63.500,A 180.000,B 0.000,C 180.000} C_DIS
LIN {X 46.060,Y 103.153,Z 63.500,A 180.000,B 0.000,C 180.000} C_DIS
LIN {X 46.145,Y 103.690,Z 63.500,A 180.000,B 0.000,C 180.000} C_DIS
LIN {X 46.176,Y 103.869,Z 63.500,A 180.000,B 0.000,C 180.000} C_DIS
LIN {X 46.215,Y 104.047,Z 63.500,A 180.000,B 0.000,C 180.000} C_DIS
LIN {X 46.305,Y 104.449,Z 63.500,A 180.000,B 0.000,C 180.000} C_DIS
LIN {X 46.335,Y 104.584,Z 63.500,A 180.000,B 0.000,C 180.000} C_DIS
LIN {X 46.384,Y 104.762,Z 63.500,A 180.000,B 0.000,C 180.000} C_DIS
LIN {X 46.540,Y 105.299,Z 63.500,A 180.000,B 0.000,C 180.000} C_DIS
LIN {X 46.599,Y 105.477,Z 63.500,A 180.000,B 0.000,C 180.000} C_DIS
LIN {X 46.792,Y 106.014,Z 63.500,A 180.000,B 0.000,C 180.000} C_DIS
LIN {X 46.841,Y 106.144,Z 63.500,A 180.000,B 0.000,C 180.000} C_DIS
LIN {X 46.861,Y 106.193,Z 63.500,A 180.000,B 0.000,C 180.000} C_DIS
LIN {X 47.093,Y 106.729,Z 63.500,A 180.000,B 0.000,C 180.000} C_DIS
LIN {X 47.176,Y 106.908,Z 63.500,A 180.000,B 0.000,C 180.000} C_DIS
LIN {X 47.198,Y 106.952,Z 63.500,A 180.000,B 0.000,C 180.000} C_DIS
LIN {X 47.449,Y 107.444,Z 63.500,A 180.000,B 0.000,C 180.000} C_DIS
LIN {X 47.546,Y 107.623,Z 63.500,A 180.000,B 0.000,C 180.000} C_DIS
LIN {X 47.863,Y 108.159,Z 63.500,A 180.000,B 0.000,C 180.000} C_DIS
LIN {X 47.914,Y 108.240,Z 63.500,A 180.000,B 0.000,C 180.000} C_DIS
LIN {X 47.979,Y 108.338,Z 63.500,A 180.000,B 0.000,C 180.000} C_DIS
LIN {X 48.271,Y 108.767,Z 63.500,A 180.000,B 0.000,C 180.000} C_DIS
LIN {X 48.345,Y 108.874,Z 63.500,A 180.000,B 0.000,C 180.000} C_DIS
LIN {X 48.450,Y 109.012,Z 63.500,A 180.000,B 0.000,C 180.000} C_DIS
LIN {X 48.759,Y 109.410,Z 63.500,A 180.000,B 0.000,C 180.000} C_DIS
LIN {X 48.807,Y 109.472,Z 63.500,A 180.000,B 0.000,C 180.000} C_DIS
LIN {X 48.907,Y 109.589,Z 63.500,A 180.000,B 0.000,C 180.000} C_DIS
LIN {X 49.223,Y 109.947,Z 63.500,A 180.000,B 0.000,C 180.000} C_DIS
LIN {X 49.344,Y 110.083,Z 63.500,A 180.000,B 0.000,C 180.000} C_DIS
LIN {X 49.384,Y 110.126,Z 63.500,A 180.000,B 0.000,C 180.000} C_DIS
LIN {X 49.523,Y 110.264,Z 63.500,A 180.000,B 0.000,C 180.000} C_DIS
LIN {X 49.742,Y 110.483,Z 63.500,A 180.000,B 0.000,C 180.000} C_DIS
LIN {X 49.880,Y 110.621,Z 63.500,A 180.000,B 0.000,C 180.000} C_DIS
LIN {X 49.923,Y 110.662,Z 63.500,A 180.000,B 0.000,C 180.000} C_DIS
LIN {X 50.059,Y 110.782,Z 63.500,A 180.000,B 0.000,C 180.000} C_DIS
LIN {X 50.416,Y 111.098,Z 63.500,A 180.000,B 0.000,C 180.000} C_DIS
LIN {X 50.535,Y 111.198,Z 63.500,A 180.000,B 0.000,C 180.000} C_DIS
LIN {X 50.595,Y 111.245,Z 63.500,A 180.000,B 0.000,C 180.000} C_DIS
LIN {X 50.996,Y 111.556,Z 63.500,A 180.000,B 0.000,C 180.000} C_DIS
LIN {X 51.131,Y 111.659,Z 63.500,A 180.000,B 0.000,C 180.000} C_DIS
LIN {X 51.241,Y 111.734,Z 63.500,A 180.000,B 0.000,C 180.000} C_DIS
LIN {X 51.668,Y 112.025,Z 63.500,A 180.000,B 0.000,C 180.000} C_DIS
LIN {X 51.769,Y 112.092,Z 63.500,A 180.000,B 0.000,C 180.000} C_DIS
LIN {X 51.847,Y 112.140,Z 63.500,A 180.000,B 0.000,C 180.000} C_DIS
LIN {X 52.383,Y 112.457,Z 63.500,A 180.000,B 0.000,C 180.000} C_DIS
LIN {X 52.562,Y 112.554,Z 63.500,A 180.000,B 0.000,C 180.000} C_DIS
LIN {X 53.059,Y 112.807,Z 63.500,A 180.000,B 0.000,C 180.000} C_DIS
LIN {X 53.098,Y 112.827,Z 63.500,A 180.000,B 0.000,C 180.000} C_DIS
LIN {X 53.277,Y 112.909,Z 63.500,A 180.000,B 0.000,C 180.000} C_DIS
LIN {X 53.813,Y 113.141,Z 63.500,A 180.000,B 0.000,C 180.000} C_DIS
LIN {X 53.870,Y 113.165,Z 63.500,A 180.000,B 0.000,C 180.000} C_DIS
LIN {X 53.992,Y 113.210,Z 63.500,A 180.000,B 0.000,C 180.000} C_DIS
LIN {X 54.528,Y 113.403,Z 63.500,A 180.000,B 0.000,C 180.000} C_DIS
LIN {X 54.707,Y 113.462,Z 63.500,A 180.000,B 0.000,C 180.000} C_DIS
LIN {X 55.243,Y 113.618,Z 63.500,A 180.000,B 0.000,C 180.000} C_DIS
LIN {X 55.422,Y 113.666,Z 63.500,A 180.000,B 0.000,C 180.000} C_DIS
LIN {X 55.575,Y 113.701,Z 63.500,A 180.000,B 0.000,C 180.000} C_DIS
LIN {X 55.958,Y 113.786,Z 63.500,A 180.000,B 0.000,C 180.000} C_DIS
LIN {X 56.137,Y 113.826,Z 63.500,A 180.000,B 0.000,C 180.000} C_DIS
LIN {X 56.316,Y 113.855,Z 63.500,A 180.000,B 0.000,C 180.000} C_DIS
LIN {X 56.852,Y 113.940,Z 63.500,A 180.000,B 0.000,C 180.000} C_DIS
LIN {X 57.031,Y 113.962,Z 63.500,A 180.000,B 0.000,C 180.000} C_DIS
LIN {X 57.567,Y 114.013,Z 63.500,A 180.000,B 0.000,C 180.000} C_DIS
LIN {X 57.746,Y 114.027,Z 63.500,A 180.000,B 0.000,C 180.000} C_DIS
LIN {X 57.925,Y 114.033,Z 63.500,A 180.000,B 0.000,C 180.000} C_DIS
LIN {X 58.282,Y 114.044,Z 63.500,A 180.000,B 0.000,C 180.000} C_DIS
LIN {X 58.461,Y 114.050,Z 63.500,A 180.000,B 0.000,C 180.000} C_DIS
LIN {X 58.640,Y 114.047,Z 63.500,A 180.000,B 0.000,C 180.000} C_DIS
LIN {X 59.176,Y 114.030,Z 63.500,A 180.000,B 0.000,C 180.000} C_DIS
LIN {X 59.355,Y 114.020,Z 63.500,A 180.000,B 0.000,C 180.000} C_DIS
LIN {X 59.534,Y 114.003,Z 63.500,A 180.000,B 0.000,C 180.000} C_DIS
LIN {X 59.891,Y 113.969,Z 63.500,A 180.000,B 0.000,C 180.000} C_DIS
LIN {X 60.070,Y 113.951,Z 63.500,A 180.000,B 0.000,C 180.000} C_DIS
LIN {X 60.249,Y 113.924,Z 63.500,A 180.000,B 0.000,C 180.000} C_DIS
LIN {X 60.606,Y 113.868,Z 63.500,A 180.000,B 0.000,C 180.000} C_DIS
LIN {X 60.785,Y 113.839,Z 63.500,A 180.000,B 0.000,C 180.000} C_DIS
LIN {X 60.964,Y 113.804,Z 63.500,A 180.000,B 0.000,C 180.000} C_DIS
LIN {X 61.500,Y 113.684,Z 63.500,A 180.000,B 0.000,C 180.000} C_DIS
LIN {X 61.679,Y 113.640,Z 63.500,A 180.000,B 0.000,C 180.000} C_DIS
LIN {X 61.858,Y 113.588,Z 63.500,A 180.000,B 0.000,C 180.000} C_DIS
LIN {X 62.215,Y 113.484,Z 63.500,A 180.000,B 0.000,C 180.000} C_DIS
LIN {X 62.394,Y 113.431,Z 63.500,A 180.000,B 0.000,C 180.000} C_DIS
LIN {X 62.573,Y 113.367,Z 63.500,A 180.000,B 0.000,C 180.000} C_DIS
LIN {X 62.930,Y 113.238,Z 63.500,A 180.000,B 0.000,C 180.000} C_DIS
LIN {X 63.109,Y 113.173,Z 63.500,A 180.000,B 0.000,C 180.000} C_DIS
LIN {X 63.130,Y 113.165,Z 63.500,A 180.000,B 0.000,C 180.000} C_DIS
LIN {X 63.288,Y 113.097,Z 63.500,A 180.000,B 0.000,C 180.000} C_DIS
LIN {X 63.645,Y 112.943,Z 63.500,A 180.000,B 0.000,C 180.000} C_DIS
LIN {X 63.824,Y 112.865,Z 63.500,A 180.000,B 0.000,C 180.000} C_DIS
LIN {X 63.941,Y 112.807,Z 63.500,A 180.000,B 0.000,C 180.000} C_DIS
LIN {X 64.360,Y 112.594,Z 63.500,A 180.000,B 0.000,C 180.000} C_DIS
LIN {X 64.539,Y 112.501,Z 63.500,A 180.000,B 0.000,C 180.000} C_DIS
LIN {X 64.630,Y 112.450,Z 63.500,A 180.000,B 0.000,C 180.000} C_DIS
LIN {X 65.075,Y 112.186,Z 63.500,A 180.000,B 0.000,C 180.000} C_DIS
LIN {X 65.231,Y 112.092,Z 63.500,A 180.000,B 0.000,C 180.000} C_DIS
LIN {X 65.254,Y 112.077,Z 63.500,A 180.000,B 0.000,C 180.000} C_DIS
LIN {X 65.433,Y 111.956,Z 63.500,A 180.000,B 0.000,C 180.000} C_DIS
LIN {X 65.791,Y 111.713,Z 63.500,A 180.000,B 0.000,C 180.000} C_DIS
LIN {X 65.969,Y 111.583,Z 63.500,A 180.000,B 0.000,C 180.000} C_DIS
LIN {X 66.327,Y 111.306,Z 63.500,A 180.000,B 0.000,C 180.000} C_DIS
LIN {X 66.465,Y 111.198,Z 63.500,A 180.000,B 0.000,C 180.000} C_DIS
LIN {X 66.506,Y 111.165,Z 63.500,A 180.000,B 0.000,C 180.000} C_DIS
LIN {X 66.672,Y 111.019,Z 63.500,A 180.000,B 0.000,C 180.000} C_DIS
LIN {X 66.875,Y 110.841,Z 63.500,A 180.000,B 0.000,C 180.000} C_DIS
LIN {X 67.042,Y 110.693,Z 63.500,A 180.000,B 0.000,C 180.000} C_DIS
LIN {X 67.077,Y 110.662,Z 63.500,A 180.000,B 0.000,C 180.000} C_DIS
LIN {X 67.221,Y 110.521,Z 63.500,A 180.000,B 0.000,C 180.000} C_DIS
LIN {X 67.578,Y 110.163,Z 63.500,A 180.000,B 0.000,C 180.000} C_DIS
LIN {X 67.616,Y 110.126,Z 63.500,A 180.000,B 0.000,C 180.000} C_DIS
LIN {X 67.757,Y 109.970,Z 63.500,A 180.000,B 0.000,C 180.000} C_DIS
LIN {X 68.115,Y 109.564,Z 63.500,A 180.000,B 0.000,C 180.000} C_DIS
LIN {X 68.241,Y 109.410,Z 63.500,A 180.000,B 0.000,C 180.000} C_DIS
LIN {X 68.518,Y 109.053,Z 63.500,A 180.000,B 0.000,C 180.000} C_DIS
LIN {X 68.651,Y 108.880,Z 63.500,A 180.000,B 0.000,C 180.000} C_DIS
LIN {X 68.655,Y 108.874,Z 63.500,A 180.000,B 0.000,C 180.000} C_DIS
LIN {X 68.778,Y 108.695,Z 63.500,A 180.000,B 0.000,C 180.000} C_DIS
LIN {X 69.021,Y 108.338,Z 63.500,A 180.000,B 0.000,C 180.000} C_DIS
LIN {X 69.137,Y 108.159,Z 63.500,A 180.000,B 0.000,C 180.000} C_DIS
LIN {X 69.454,Y 107.623,Z 63.500,A 180.000,B 0.000,C 180.000} C_DIS
LIN {X 69.545,Y 107.456,Z 63.500,A 180.000,B 0.000,C 180.000} C_DIS
LIN {X 69.733,Y 107.086,Z 63.500,A 180.000,B 0.000,C 180.000} C_DIS
LIN {X 69.824,Y 106.908,Z 63.500,A 180.000,B 0.000,C 180.000} C_DIS
LIN {X 69.902,Y 106.739,Z 63.500,A 180.000,B 0.000,C 180.000} C_DIS
LIN {X 70.139,Y 106.193,Z 63.500,A 180.000,B 0.000,C 180.000} C_DIS
LIN {X 70.208,Y 106.014,Z 63.500,A 180.000,B 0.000,C 180.000} C_DIS
LIN {X 70.401,Y 105.477,Z 63.500,A 180.000,B 0.000,C 180.000} C_DIS
LIN {X 70.439,Y 105.369,Z 63.500,A 180.000,B 0.000,C 180.000} C_DIS
LIN {X 70.460,Y 105.299,Z 63.500,A 180.000,B 0.000,C 180.000} C_DIS
LIN {X 70.617,Y 104.758,Z 63.500,A 180.000,B 0.000,C 180.000} C_DIS
LIN {X 70.665,Y 104.584,Z 63.500,A 180.000,B 0.000,C 180.000} C_DIS
LIN {X 70.705,Y 104.405,Z 63.500,A 180.000,B 0.000,C 180.000} C_DIS
LIN {X 70.796,Y 103.999,Z 63.500,A 180.000,B 0.000,C 180.000} C_DIS
LIN {X 70.824,Y 103.869,Z 63.500,A 180.000,B 0.000,C 180.000} C_DIS
LIN {X 70.855,Y 103.690,Z 63.500,A 180.000,B 0.000,C 180.000} C_DIS
LIN {X 70.940,Y 103.153,Z 63.500,A 180.000,B 0.000,C 180.000} C_DIS
LIN {X 70.962,Y 102.975,Z 63.500,A 180.000,B 0.000,C 180.000} C_DIS
LIN {X 71.012,Y 102.438,Z 63.500,A 180.000,B 0.000,C 180.000} C_DIS
LIN {X 71.027,Y 102.260,Z 63.500,A 180.000,B 0.000,C 180.000} C_DIS
LIN {X 71.033,Y 102.081,Z 63.500,A 180.000,B 0.000,C 180.000} C_DIS
LIN {X 71.044,Y 101.723,Z 63.500,A 180.000,B 0.000,C 180.000} C_DIS
LIN {X 71.050,Y 101.545,Z 63.500,A 180.000,B 0.000,C 180.000} C_DIS
LIN {X 71.047,Y 101.366,Z 63.500,A 180.000,B 0.000,C 180.000} C_DIS
LIN {X 71.030,Y 100.829,Z 63.500,A 180.000,B 0.000,C 180.000} C_DIS
LIN {X 71.021,Y 100.651,Z 63.500,A 180.000,B 0.000,C 180.000} C_DIS
LIN {X 71.004,Y 100.472,Z 63.500,A 180.000,B 0.000,C 180.000} C_DIS
LIN {X 70.970,Y 100.114,Z 63.500,A 180.000,B 0.000,C 180.000} C_DIS
LIN {X 70.952,Y 99.936,Z 63.500,A 180.000,B 0.000,C 180.000} C_DIS
LIN {X 70.925,Y 99.757,Z 63.500,A 180.000,B 0.000,C 180.000} C_DIS
LIN {X 70.840,Y 99.221,Z 63.500,A 180.000,B 0.000,C 180.000} C_DIS
LIN {X 70.805,Y 99.042,Z 63.500,A 180.000,B 0.000,C 180.000} C_DIS
LIN {X 70.718,Y 98.654,Z 63.500,A 180.000,B 0.000,C 180.000} C_DIS
LIN {X 70.685,Y 98.505,Z 63.500,A 180.000,B 0.000,C 180.000} C_DIS
LIN {X 70.642,Y 98.327,Z 63.500,A 180.000,B 0.000,C 180.000} C_DIS
LIN {X 70.617,Y 98.242,Z 63.500,A 180.000,B 0.000,C 180.000} C_DIS
LIN {X 70.486,Y 97.790,Z 63.500,A 180.000,B 0.000,C 180.000} C_DIS
LIN {X 70.439,Y 97.631,Z 63.500,A 180.000,B 0.000,C 180.000} C_DIS
LIN {X 70.432,Y 97.612,Z 63.500,A 180.000,B 0.000,C 180.000} C_DIS
LIN {X 70.369,Y 97.433,Z 63.500,A 180.000,B 0.000,C 180.000} C_DIS
LIN {X 70.240,Y 97.075,Z 63.500,A 180.000,B 0.000,C 180.000} C_DIS
LIN {X 70.175,Y 96.897,Z 63.500,A 180.000,B 0.000,C 180.000} C_DIS
LIN {X 70.100,Y 96.718,Z 63.500,A 180.000,B 0.000,C 180.000} C_DIS
LIN {X 69.902,Y 96.261,Z 63.500,A 180.000,B 0.000,C 180.000} C_DIS
LIN {X 69.867,Y 96.181,Z 63.500,A 180.000,B 0.000,C 180.000} C_DIS
LIN {X 69.779,Y 96.003,Z 63.500,A 180.000,B 0.000,C 180.000} C_DIS
LIN {X 69.545,Y 95.544,Z 63.500,A 180.000,B 0.000,C 180.000} C_DIS
LIN {X 69.504,Y 95.466,Z 63.500,A 180.000,B 0.000,C 180.000} C_DIS
LIN {X 69.401,Y 95.288,Z 63.500,A 180.000,B 0.000,C 180.000} C_DIS
LIN {X 69.187,Y 94.927,Z 63.500,A 180.000,B 0.000,C 180.000} C_DIS
LIN {X 69.081,Y 94.751,Z 63.500,A 180.000,B 0.000,C 180.000} C_DIS
LIN {X 69.008,Y 94.644,Z 63.500,A 180.000,B 0.000,C 180.000} C_DIS
LIN {X 68.717,Y 94.215,Z 63.500,A 180.000,B 0.000,C 180.000} C_DIS
LIN {X 68.651,Y 94.120,Z 63.500,A 180.000,B 0.000,C 180.000} C_DIS
LIN {X 68.587,Y 94.036,Z 63.500,A 180.000,B 0.000,C 180.000} C_DIS
LIN {X 68.293,Y 93.657,Z 63.500,A 180.000,B 0.000,C 180.000} C_DIS
LIN {X 68.170,Y 93.500,Z 63.500,A 180.000,B 0.000,C 180.000} C_DIS
LIN {X 68.115,Y 93.436,Z 63.500,A 180.000,B 0.000,C 180.000} C_DIS
LIN {X 67.698,Y 92.964,Z 63.500,A 180.000,B 0.000,C 180.000} C_DIS
LIN {X 67.578,Y 92.837,Z 63.500,A 180.000,B 0.000,C 180.000} C_DIS
LIN {X 67.169,Y 92.427,Z 63.500,A 180.000,B 0.000,C 180.000} C_DIS
LIN {X 67.061,Y 92.325,Z 63.500,A 180.000,B 0.000,C 180.000} C_DIS
; Link Move Starts
LIN {X 66.826,Y 92.116,Z 63.500,A 180.000,B 0.000,C 180.000} C_DIS
LIN {X 66.589,Y 91.907,Z 63.499,A 180.000,B 0.000,C 180.000} C_DIS
LIN {X 66.345,Y 91.709,Z 63.498,A 180.000,B 0.000,C 180.000} C_DIS
LIN {X 66.096,Y 91.516,Z 63.496,A 180.000,B 0.000,C 180.000} C_DIS
LIN {X 65.846,Y 91.325,Z 63.494,A 180.000,B 0.000,C 180.000} C_DIS
LIN {X 65.585,Y 91.147,Z 63.491,A 180.000,B 0.000,C 180.000} C_DIS
LIN {X 65.325,Y 90.970,Z 63.488,A 180.000,B 0.000,C 180.000} C_DIS
LIN {X 65.058,Y 90.804,Z 63.485,A 180.000,B 0.000,C 180.000} C_DIS
LIN {X 64.787,Y 90.643,Z 63.481,A 180.000,B 0.000,C 180.000} C_DIS
LIN {X 64.514,Y 90.485,Z 63.477,A 180.000,B 0.000,C 180.000} C_DIS
LIN {X 64.234,Y 90.342,Z 63.472,A 180.000,B 0.000,C 180.000} C_DIS
LIN {X 64.093,Y 90.270,Z 63.469,A 180.000,B 0.000,C 180.000} C_DIS
LIN {X 63.953,Y 90.199,Z 63.467,A 180.000,B 0.000,C 180.000} C_DIS
LIN {X 63.811,Y 90.130,Z 63.464,A 180.000,B 0.000,C 180.000} C_DIS
LIN {X 63.667,Y 90.067,Z 63.461,A 180.000,B 0.000,C 180.000} C_DIS
LIN {X 63.523,Y 90.004,Z 63.459,A 180.000,B 0.000,C 180.000} C_DIS
LIN {X 63.378,Y 89.942,Z 63.456,A 180.000,B 0.000,C 180.000} C_DIS
LIN {X 63.233,Y 89.879,Z 63.452,A 180.000,B 0.000,C 180.000} C_DIS
LIN {X 63.088,Y 89.819,Z 63.449,A 180.000,B 0.000,C 180.000} C_DIS
LIN {X 62.940,Y 89.765,Z 63.446,A 180.000,B 0.000,C 180.000} C_DIS
LIN {X 62.792,Y 89.712,Z 63.443,A 180.000,B 0.000,C 180.000} C_DIS
LIN {X 62.643,Y 89.658,Z 63.439,A 180.000,B 0.000,C 180.000} C_DIS
LIN {X 62.495,Y 89.605,Z 63.436,A 180.000,B 0.000,C 180.000} C_DIS
LIN {X 62.346,Y 89.554,Z 63.432,A 180.000,B 0.000,C 180.000} C_DIS
LIN {X 62.195,Y 89.510,Z 63.428,A 180.000,B 0.000,C 180.000} C_DIS
LIN {X 62.044,Y 89.466,Z 63.425,A 180.000,B 0.000,C 180.000} C_DIS
LIN {X 61.893,Y 89.422,Z 63.421,A 180.000,B 0.000,C 180.000} C_DIS
LIN {X 61.741,Y 89.378,Z 63.417,A 180.000,B 0.000,C 180.000} C_DIS
LIN {X 61.589,Y 89.336,Z 63.413,A 180.000,B 0.000,C 180.000} C_DIS
LIN {X 61.436,Y 89.302,Z 63.409,A 180.000,B 0.000,C 180.000} C_DIS
LIN {X 61.282,Y 89.267,Z 63.405,A 180.000,B 0.000,C 180.000} C_DIS
LIN {X 61.128,Y 89.233,Z 63.400,A 180.000,B 0.000,C 180.000} C_DIS
LIN {X 60.975,Y 89.199,Z 63.396,A 180.000,B 0.000,C 180.000} C_DIS
LIN {X 60.820,Y 89.167,Z 63.392,A 180.000,B 0.000,C 180.000} C_DIS
LIN {X 60.665,Y 89.141,Z 63.387,A 180.000,B 0.000,C 180.000} C_DIS
LIN {X 60.509,Y 89.117,Z 63.383,A 180.000,B 0.000,C 180.000} C_DIS
LIN {X 60.354,Y 89.092,Z 63.378,A 180.000,B 0.000,C 180.000} C_DIS
LIN {X 60.198,Y 89.068,Z 63.373,A 180.000,B 0.000,C 180.000} C_DIS
LIN {X 60.042,Y 89.045,Z 63.369,A 180.000,B 0.000,C 180.000} C_DIS
LIN {X 59.886,Y 89.030,Z 63.364,A 180.000,B 0.000,C 180.000} C_DIS
LIN {X 59.729,Y 89.015,Z 63.359,A 180.000,B 0.000,C 180.000} C_DIS
LIN {X 59.572,Y 89.000,Z 63.354,A 180.000,B 0.000,C 180.000} C_DIS
LIN {X 59.494,Y 88.993,Z 63.351,A 180.000,B 0.000,C 180.000} C_DIS
LIN {X 59.415,Y 88.986,Z 63.349,A 180.000,B 0.000,C 180.000} C_DIS
LIN {X 59.337,Y 88.978,Z 63.346,A 180.000,B 0.000,C 180.000} C_DIS
LIN {X 59.258,Y 88.973,Z 63.344,A 180.000,B 0.000,C 180.000} C_DIS
LIN {X 59.180,Y 88.970,Z 63.341,A 180.000,B 0.000,C 180.000} C_DIS
LIN {X 59.101,Y 88.968,Z 63.339,A 180.000,B 0.000,C 180.000} C_DIS
LIN {X 59.022,Y 88.965,Z 63.336,A 180.000,B 0.000,C 180.000} C_DIS
LIN {X 58.865,Y 88.960,Z 63.331,A 180.000,B 0.000,C 180.000} C_DIS
LIN {X 58.707,Y 88.955,Z 63.325,A 180.000,B 0.000,C 180.000} C_DIS
LIN {X 58.629,Y 88.953,Z 63.323,A 180.000,B 0.000,C 180.000} C_DIS
LIN {X 58.550,Y 88.950,Z 63.320,A 180.000,B 0.000,C 180.000} C_DIS
LIN {X 58.471,Y 88.950,Z 63.317,A 180.000,B 0.000,C 180.000} C_DIS
LIN {X 58.392,Y 88.952,Z 63.315,A 180.000,B 0.000,C 180.000} C_DIS
LIN {X 58.235,Y 88.957,Z 63.309,A 180.000,B 0.000,C 180.000} C_DIS
LIN {X 58.156,Y 88.960,Z 63.306,A 180.000,B 0.000,C 180.000} C_DIS
LIN {X 57.999,Y 88.965,Z 63.301,A 180.000,B 0.000,C 180.000} C_DIS
LIN {X 57.841,Y 88.969,Z 63.296,A 180.000,B 0.000,C 180.000} C_DIS
LIN {X 57.763,Y 88.972,Z 63.293,A 180.000,B 0.000,C 180.000} C_DIS
LIN {X 57.684,Y 88.977,Z 63.290,A 180.000,B 0.000,C 180.000} C_DIS
LIN {X 57.606,Y 88.984,Z 63.287,A 180.000,B 0.000,C 180.000} C_DIS
LIN {X 57.527,Y 88.991,Z 63.285,A 180.000,B 0.000,C 180.000} C_DIS
LIN {X 57.370,Y 89.006,Z 63.279,A 180.000,B 0.000,C 180.000} C_DIS
LIN {X 57.135,Y 89.028,Z 63.271,A 180.000,B 0.000,C 180.000} C_DIS
LIN {X 57.057,Y 89.035,Z 63.268,A 180.000,B 0.000,C 180.000} C_DIS
LIN {X 56.978,Y 89.043,Z 63.265,A 180.000,B 0.000,C 180.000} C_DIS
LIN {X 56.900,Y 89.052,Z 63.263,A 180.000,B 0.000,C 180.000} C_DIS
LIN {X 56.822,Y 89.064,Z 63.260,A 180.000,B 0.000,C 180.000} C_DIS
LIN {X 56.667,Y 89.089,Z 63.254,A 180.000,B 0.000,C 180.000} C_DIS
LIN {X 56.589,Y 89.101,Z 63.252,A 180.000,B 0.000,C 180.000} C_DIS
LIN {X 56.433,Y 89.126,Z 63.246,A 180.000,B 0.000,C 180.000} C_DIS
LIN {X 56.278,Y 89.151,Z 63.241,A 180.000,B 0.000,C 180.000} C_DIS
LIN {X 56.200,Y 89.163,Z 63.238,A 180.000,B 0.000,C 180.000} C_DIS
LIN {X 56.123,Y 89.177,Z 63.235,A 180.000,B 0.000,C 180.000} C_DIS
LIN {X 56.046,Y 89.194,Z 63.232,A 180.000,B 0.000,C 180.000} C_DIS
LIN {X 55.969,Y 89.211,Z 63.230,A 180.000,B 0.000,C 180.000} C_DIS
LIN {X 55.815,Y 89.246,Z 63.224,A 180.000,B 0.000,C 180.000} C_DIS
LIN {X 55.508,Y 89.314,Z 63.213,A 180.000,B 0.000,C 180.000} C_DIS
